//-------SIGNAL -> X_E_Tot_Cosu Max: 4.29497e+08 Min: 0 Def: 0 Resolution: 0.1 Offset: 0
GVL.IOVD.X_E_Tot_Cosu.v						:= GVL.SY.S_ECU_Rdy AND NOT GVL.IOVD.X_E_Tot_Cosu.e	AND NOT GVL.IOVD.X_E_Tot_Cosu.na AND NOT GVL.IOVD.X_E_Tot_Cosu.RangeExcd;
GVL.IOVD.X_E_Tot_Cosu.x						:= GVL.PV.X_E_Tot_Cosu;
GVL.IOVD.X_E_Tot_Cosu.e						:= FALSE;
GVL.IOVD.X_E_Tot_Cosu.na					:= FALSE;
GVL.IOVD.X_E_Tot_Cosu.RangeExcd				:= (429496729.4 < GVL.IOVD.X_E_Tot_Cosu.x) OR (0 > GVL.IOVD.X_E_Tot_Cosu.x);	 
//-------SIGNAL -> X_Avg_Cosu_Opp Max: 65,535 Min: 0 Def: 0 Resolution: 0.1 Offset: 0
GVL.IOVD.X_Avg_Cosu_Opp.v					:= GVL.SY.S_ECU_Rdy AND NOT GVL.IOVD.X_Avg_Cosu_Opp.e	AND NOT GVL.IOVD.X_Avg_Cosu_Opp.na AND NOT GVL.IOVD.X_Avg_Cosu_Opp.RangeExcd;
GVL.IOVD.X_Avg_Cosu_Opp.x					:= GVL.PV.X_Avg_Cosu_Opp;
GVL.IOVD.X_Avg_Cosu_Opp.e					:= FALSE;
GVL.IOVD.X_Avg_Cosu_Opp.na					:= FALSE;
GVL.IOVD.X_Avg_Cosu_Opp.RangeExcd			:= (65.535 < GVL.IOVD.X_Avg_Cosu_Opp.x) OR (0 > GVL.IOVD.X_Avg_Cosu_Opp.x);		  
{endregion}
//-----------------------------------------------------------------------------------------------------------------------------
//-----------------------------------------------------------------------------------------------------------------------------
//MESSAGE------
{region " User Area : Arac_Genel_Istatistik_2- ID:4C9"}

//-------SIGNAL -> X_Daily_Avg_Cosu Max: 40 Min: 0 Def: 0 Resolution: 0.001 Offset: 0
GVL.IOVD.X_Daily_Avg_Cosu.v					:= GVL.SY.S_ECU_Rdy AND NOT GVL.IOVD.X_Daily_Avg_Cosu.e	AND NOT GVL.IOVD.X_Daily_Avg_Cosu.na AND NOT GVL.IOVD.X_Daily_Avg_Cosu.RangeExcd;
GVL.IOVD.X_Daily_Avg_Cosu.x					:= GVL.PV.X_Avg_Cosu;
GVL.IOVD.X_Daily_Avg_Cosu.e					:= FALSE;
GVL.IOVD.X_Daily_Avg_Cosu.na				:= FALSE;
GVL.IOVD.X_Daily_Avg_Cosu.RangeExcd			:= (40 < GVL.IOVD.X_Daily_Avg_Cosu.x) OR (0 > GVL.IOVD.X_Daily_Avg_Cosu.x);
//-------SIGNAL -> X_Trp_Distn Max: 4.21108e+08 Min: 0 Def: 0 Resolution: 0.1 Offset: 0
GVL.IOVD.X_Trp_Distn.v						:= GVL.SY.S_ECU_Rdy AND NOT GVL.IOVD.X_Trp_Distn.e	AND NOT GVL.IOVD.X_Trp_Distn.na AND NOT GVL.IOVD.X_Trp_Distn.RangeExcd;
GVL.IOVD.X_Trp_Distn.x						:= GVL.PV.X_Trp_Bat;
GVL.IOVD.X_Trp_Distn.e						:= FALSE;
GVL.IOVD.X_Trp_Distn.na						:= FALSE;
GVL.IOVD.X_Trp_Distn.RangeExcd				:= (421108121.5 < GVL.IOVD.X_Trp_Distn.x) OR (0 > GVL.IOVD.X_Trp_Distn.x);
//-------SIGNAL -> X_U_ECU_Sp Max: 100 Min: 0 Def: 0 Resolution: 1 Offset: 0
GVL.IOVD.X_U_ECU_Sp.v						:= GVL.SY.S_ECU_Rdy AND NOT GVL.IOVD.X_U_ECU_Sp.e	AND NOT GVL.IOVD.X_U_ECU_Sp.na AND NOT GVL.IOVD.X_U_ECU_Sp.RangeExcd;
GVL.IOVD.X_U_ECU_Sp.x						:= ANY_TO_REAL(GVL.IC.X_U_Bat.value);
GVL.IOVD.X_U_ECU_Sp.e						:= FALSE;
GVL.IOVD.X_U_ECU_Sp.na						:= FALSE;
GVL.IOVD.X_U_ECU_Sp.RangeExcd				:= (40000 < GVL.IOVD.X_U_ECU_Sp.x )OR (0 > GVL.IOVD.X_U_ECU_Sp.x);		
{endregion}
//-----------------------------------------------------------------------------------------------------------------------------
//-----------------------------------------------------------------------------------------------------------------------------
//MESSAGE------
{region " User Area : Klima_Calisma_Sureleri_1- ID:4CA"}

//-------SIGNAL -> N_Hvac_Drv_Op_Cnt Max: 4.29497e+09 Min: 0 Def: 0 Resolution: 1 Offset: 0
GVL.IOVD.N_Hvac_Drv_Op_Cnt.v				:= GVL.SY.S_ECU_Rdy AND NOT GVL.IOVD.N_Hvac_Drv_Op_Cnt.e AND NOT GVL.IOVD.N_Hvac_Drv_Op_Cnt.na AND NOT GVL.IOVD.N_Hvac_Drv_Op_Cnt.RangeExcd;
GVL.IOVD.N_Hvac_Drv_Op_Cnt.x				:= DINT_TO_UDINT(TRUNC(GVL.PV.X_Tm_Tot_HVAC_Drv_Op / 60));		// PR1006_REV_002637_TIMTRO
GVL.IOVD.N_Hvac_Drv_Op_Cnt.e				:= FALSE;
GVL.IOVD.N_Hvac_Drv_Op_Cnt.na				:= FALSE;
GVL.IOVD.N_Hvac_Drv_Op_Cnt.RangeExcd		:= (4294967294 < GVL.IOVD.N_Hvac_Drv_Op_Cnt.x) OR (0 > GVL.IOVD.N_Hvac_Drv_Op_Cnt.x);
//-------SIGNAL -> N_Hvac_Pass1_Op_Cnt Max: 4.29497e+09 Min: 0 Def: 0 Resolution: 1 Offset: 0
GVL.IOVD.N_Hvac_Pass1_Op_Cnt.v				:= GVL.SY.S_ECU_Rdy AND NOT GVL.IOVD.N_Hvac_Pass1_Op_Cnt.e	AND NOT GVL.IOVD.N_Hvac_Pass1_Op_Cnt.na AND NOT GVL.IOVD.N_Hvac_Pass1_Op_Cnt.RangeExcd;
GVL.IOVD.N_Hvac_Pass1_Op_Cnt.x				:= DINT_TO_UDINT(TRUNC(GVL.PV.X_Tm_Tot_HVAC_Pass1_Op / 60));	// PR1006_REV_002637_TIMTRO
GVL.IOVD.N_Hvac_Pass1_Op_Cnt.e				:= FALSE;
GVL.IOVD.N_Hvac_Pass1_Op_Cnt.na				:= FALSE;
GVL.IOVD.N_Hvac_Pass1_Op_Cnt.RangeExcd		:= (4294967294 < GVL.IOVD.N_Hvac_Pass1_Op_Cnt.x) OR (0 > GVL.IOVD.N_Hvac_Pass1_Op_Cnt.x);
{endregion}
//-----------------------------------------------------------------------------------------------------------------------------
//-----------------------------------------------------------------------------------------------------------------------------
//MESSAGE------
{region " User Area : Klima_Calisma_Sureleri_2- ID:4CB"}

//-------SIGNAL -> N_Hvac_Pass2_Op_Cnt Max: 4.29497e+09 Min: 0 Def: 0 Resolution: 1 Offset: 0
GVL.IOVD.N_Hvac_Pass2_Op_Cnt.v				:= GVL.SY.S_ECU_Rdy AND NOT GVL.IOVD.N_Hvac_Pass2_Op_Cnt.e	AND NOT GVL.IOVD.N_Hvac_Pass2_Op_Cnt.na AND NOT GVL.IOVD.N_Hvac_Pass2_Op_Cnt.RangeExcd;
GVL.IOVD.N_Hvac_Pass2_Op_Cnt.x				:= T_N_Hvac_Pass2_Op_Cnt; //eklenecek
GVL.IOVD.N_Hvac_Pass2_Op_Cnt.e				:= FALSE;
GVL.IOVD.N_Hvac_Pass2_Op_Cnt.na				:= FALSE;
GVL.IOVD.N_Hvac_Pass2_Op_Cnt.RangeExcd		:= (4294967294 < GVL.IOVD.N_Hvac_Pass2_Op_Cnt.x) OR (0 > GVL.IOVD.N_Hvac_Pass2_Op_Cnt.x);
//-------SIGNAL -> N_Btms_Op_Cnt Max: 4.29497e+09 Min: 0 Def: 0 Resolution: 1 Offset: 0
GVL.IOVD.N_Btms_Op_Cnt.v					:= GVL.SY.S_ECU_Rdy AND NOT GVL.IOVD.N_Btms_Op_Cnt.e AND NOT GVL.IOVD.N_Btms_Op_Cnt.na AND NOT GVL.IOVD.N_Btms_Op_Cnt.RangeExcd;
GVL.IOVD.N_Btms_Op_Cnt.x					:= REAL_TO_UDINT(GVL.PV.X_Tm_Tot_BTMS_Op); // PR1006_REV_002446_TIMTRO
GVL.IOVD.N_Btms_Op_Cnt.e					:= FALSE;
GVL.IOVD.N_Btms_Op_Cnt.na					:= FALSE;
GVL.IOVD.N_Btms_Op_Cnt.RangeExcd			:= (4294967294 < GVL.IOVD.N_Btms_Op_Cnt.x) OR (0 > GVL.IOVD.N_Btms_Op_Cnt.x);
{endregion}
//-----------------------------------------------------------------------------------------------------------------------------
//-----------------------------------------------------------------------------------------------------------------------------
//MESSAGE------
{region " User Area : Sayicilar_1- ID:4CC"}

// PR1006_REV_002519_TIMTRO
//-------SIGNAL -> N_Air_Cmp_Op_Cnt Max: 4.29497e+09 Min: 0 Def: 0 Resolution: 1 Offset: 0
GVL.IOVD.N_Air_Cmp_Op_Cnt.v					:= GVL.SY.S_ECU_Rdy AND NOT GVL.IOVD.N_Air_Cmp_Op_Cnt.e	AND NOT GVL.IOVD.N_Air_Cmp_Op_Cnt.na AND NOT GVL.IOVD.N_Air_Cmp_Op_Cnt.RangeExcd;
GVL.IOVD.N_Air_Cmp_Op_Cnt.x					:= REAL_TO_UDINT(GVL.PV.X_Tm_Tot_Air_Cmp_Op);
GVL.IOVD.N_Air_Cmp_Op_Cnt.e					:= FALSE;
GVL.IOVD.N_Air_Cmp_Op_Cnt.na					:= FALSE;
GVL.IOVD.N_Air_Cmp_Op_Cnt.RangeExcd			:= (4294967294 < GVL.IOVD.N_Air_Cmp_Op_Cnt.x) OR (0 > GVL.IOVD.N_Air_Cmp_Op_Cnt.x);
//-------SIGNAL -> X_Opp_Dist_Bat Max: 6535.5 Min: 0 Def: 0 Resolution: 1 Offset: 0
GVL.IOVD.X_Opp_Dist_Bat.v					:= GVL.SY.S_ECU_Rdy AND NOT GVL.IOVD.X_Opp_Dist_Bat.e	AND NOT GVL.IOVD.X_Opp_Dist_Bat.na AND NOT GVL.IOVD.X_Opp_Dist_Bat.RangeExcd;
GVL.IOVD.X_Opp_Dist_Bat.x					:= GVL.PV.X_Opp_Dist_Bat;
GVL.IOVD.X_Opp_Dist_Bat.e					:= FALSE;
GVL.IOVD.X_Opp_Dist_Bat.na					:= FALSE;
GVL.IOVD.X_Opp_Dist_Bat.RangeExcd			:= (6553.5 < GVL.IOVD.X_Opp_Dist_Bat.x ) OR (0 > GVL.IOVD.X_Opp_Dist_Bat.x);	 		  
{endregion}
//-----------------------------------------------------------------------------------------------------------------------------
//-----------------------------------------------------------------------------------------------------------------------------
//MESSAGE------
{region " User Area : Yardimci_Tuketici_Enerjileri- ID:4CD"}

//-------SIGNAL -> X_E_Aux_Cons Max: 4.29497e+08 Min: 0 Def: 0 Resolution: 0.1 Offset: 0
GVL.IOVD.X_E_Aux_Cons.v						:= GVL.SY.S_ECU_Rdy AND NOT GVL.IOVD.X_E_Aux_Cons.e	AND NOT GVL.IOVD.X_E_Aux_Cons.na AND NOT GVL.IOVD.X_E_Aux_Cons.RangeExcd;
GVL.IOVD.X_E_Aux_Cons.x						:= (GVL.PV.X_E_Tot_Aux_AC + GVL.PV.X_E_Tot_Aux_DC + GVL.PV.X_E_Tot_Aux_DC_24V) / 100;
GVL.IOVD.X_E_Aux_Cons.e						:= FALSE;
GVL.IOVD.X_E_Aux_Cons.na					:= FALSE;
GVL.IOVD.X_E_Aux_Cons.RangeExcd				:= (429496729.4 < GVL.IOVD.X_E_Aux_Cons.x ) OR (0 > GVL.IOVD.X_E_Aux_Cons.x);
//-------SIGNAL -> X_E_Aux_Hvac_Cons Max: 4.29497e+08 Min: 0 Def: 0 Resolution: 0.1 Offset: 0
GVL.IOVD.X_E_Aux_Hvac_Cons.v				:= GVL.SY.S_ECU_Rdy AND NOT GVL.IOVD.X_E_Cosu.e	AND NOT GVL.IOVD.X_E_Cosu.na AND NOT GVL.IOVD.X_E_Cosu.RangeExcd;
GVL.IOVD.X_E_Aux_Hvac_Cons.x				:= GVL.PV.X_E_Tot_Aux_DC / 100;
GVL.IOVD.X_E_Aux_Hvac_Cons.e				:= FALSE;
GVL.IOVD.X_E_Aux_Hvac_Cons.na				:= FALSE;
GVL.IOVD.X_E_Aux_Hvac_Cons.RangeExcd		:= (429496729.4 < GVL.IOVD.X_E_Aux_Hvac_Cons.x ) OR (0 > GVL.IOVD.X_E_Aux_Hvac_Cons.x);
{endregion}
//-----------------------------------------------------------------------------------------------------------------------------
//-----------------------------------------------------------------------------------------------------------------------------
//-----------------------------------------------------------------------------------------------------------------------------
//MESSAGE------
{region " User Area : Kapi_Sayicilari_1- ID:4CE"}

//-------SIGNAL -> N_Dr1_Cycle Max: 4.29497e+09 Min: 0 Def: 0 Resolution: 1 Offset: 0
GVL.IOVD.N_Dr1_Cycle.v					:= GVL.SY.S_ECU_Rdy AND NOT GVL.IOVD.N_Dr1_Cycle.RangeExcd;
GVL.IOVD.N_Dr1_Cycle.x					:= GVL.PV.N_Dr1_Cyc;
GVL.IOVD.N_Dr1_Cycle.RangeExcd			:= (4294967294 < GVL.IOVD.N_Dr1_Cycle.x) OR (0 > GVL.IOVD.N_Dr1_Cycle.x);
//-------SIGNAL -> N_Dr2_Cycle Max: 4.29497e+09 Min: 0 Def: 0 Resolution: 1 Offset: 0
GVL.IOVD.N_Dr2_Cycle.v					:= GVL.SY.S_ECU_Rdy AND NOT GVL.IOVD.N_Dr2_Cycle.RangeExcd;
GVL.IOVD.N_Dr2_Cycle.x					:= GVL.PV.N_Dr2_Cyc;
GVL.IOVD.N_Dr2_Cycle.RangeExcd			:= (4294967294 < GVL.IOVD.N_Dr2_Cycle.x) OR (0 > GVL.IOVD.N_Dr2_Cycle.x);
{endregion}
//-----------------------------------------------------------------------------------------------------------------------------
//-----------------------------------------------------------------------------------------------------------------------------
//MESSAGE------
{region " User Area : Kapi_Sayicilari_2- ID:4CE"}

//-------SIGNAL -> N_Dr3_Cycle Max: 4.29497e+09 Min: 0 Def: 0 Resolution: 1 Offset: 0
GVL.IOVD.N_Dr3_Cycle.v					:= GVL.SY.S_ECU_Rdy AND NOT GVL.IOVD.N_Dr3_Cycle.RangeExcd;
GVL.IOVD.N_Dr3_Cycle.x					:= GVL.PV.N_Dr3_Cyc;
GVL.IOVD.N_Dr3_Cycle.RangeExcd			:= (4294967294 < GVL.IOVD.N_Dr3_Cycle.x) OR (0 > GVL.IOVD.N_Dr3_Cycle.x);
//-------SIGNAL -> N_Dr4_Cycle Max: 4.29497e+09 Min: 0 Def: 0 Resolution: 1 Offset: 0
GVL.IOVD.N_Dr4_Cycle.v					:= GVL.SY.S_ECU_Rdy AND NOT GVL.IOVD.N_Dr4_Cycle.RangeExcd;
GVL.IOVD.N_Dr4_Cycle.x					:= 0;
GVL.IOVD.N_Dr4_Cycle.RangeExcd			:= (4294967294 < GVL.IOVD.N_Dr4_Cycle.x) OR (0 > GVL.IOVD.N_Dr4_Cycle.x);
{endregion}
//-----------------------------------------------------------------------------------------------------------------------------
//-----------------------------------------------------------------------------------------------------------------------------
//MESSAGE------
{region " User Area : Sarj_Enerjisi- ID:4D0"}

//-------SIGNAL -> X_E_Chrg_Pan Max: 4.29497e+08 Min: 0 Def: 0 Resolution: 0.1 Offset: 0
GVL.IOVD.X_E_Chrg_Pan.v					:= GVL.SY.S_ECU_Rdy AND NOT GVL.IOVD.X_E_Chrg_Pan.RangeExcd;
GVL.IOVD.X_E_Chrg_Pan.x					:= GVL.PV.X_E_Pnt_Chrg_Cosu;
GVL.IOVD.X_E_Chrg_Pan.RangeExcd			:= (429496729.4 < GVL.IOVD.X_E_Chrg_Pan.x) OR (0 > GVL.IOVD.X_E_Chrg_Pan.x);
//-------SIGNAL -> X_E_Chrg_Onbrd Max: 4.29497e+08 Min: 0 Def: 0 Resolution: 0.1 Offset: 0
GVL.IOVD.X_E_Chrg_Onbrd.v				:= GVL.SY.S_ECU_Rdy AND NOT GVL.IOVD.X_E_Chrg_Onbrd.RangeExcd;
GVL.IOVD.X_E_Chrg_Onbrd.x				:= GVL.PV.X_E_Ser_Chrg_Cosu;
GVL.IOVD.X_E_Chrg_Onbrd.RangeExcd		:= (429496729.4 < GVL.IOVD.X_E_Chrg_Onbrd.x) OR (0 > GVL.IOVD.X_E_Chrg_Onbrd.x);
{endregion}
//-----------------------------------------------------------------------------------------------------------------------------
//-----------------------------------------------------------------------------------------------------------------------------

//MESSAGE------
{region " User Area : Arac_Bilgi_1- ID:4E0"}

//-------SIGNAL -> X_Vh_No Max: 65000 Min: 0 Def: 0 Resolution: 1 Offset: 0
GVL.IOVD.X_Vh_No.v						:= GVL.SY.S_ECU_Rdy AND NOT GVL.IOVD.X_Vh_No.e AND NOT GVL.IOVD.X_Vh_No.na AND NOT GVL.IOVD.X_Vh_No.RangeExcd;
GVL.IOVD.X_Vh_No.x						:= GVL.PV.X_Vh_No;
GVL.IOVD.X_Vh_No.e						:= FALSE;
GVL.IOVD.X_Vh_No.na						:= FALSE;
GVL.IOVD.X_Vh_No.RangeExcd				:= (65000 < GVL.IOVD.X_Vh_No.x) OR (0 > GVL.IOVD.X_Vh_No.x);
//-------SIGNAL -> X_Sw_Ver_Mjr_ECU Max: 250 Min: 0 Def: 0 Resolution: 1 Offset: 0
GVL.IOVD.X_Sw_Ver_Mjr_ECU.v				:= GVL.SY.S_ECU_Rdy AND NOT GVL.IOVD.X_Sw_Ver_Mjr_ECU.e	AND NOT GVL.IOVD.X_Sw_Ver_Mjr_ECU.na AND NOT GVL.IOVD.X_Sw_Ver_Mjr_ECU.RangeExcd;
GVL.IOVD.X_Sw_Ver_Mjr_ECU.x				:= GVL.IC.X_Sw_Ver_Mjr_ECU;
GVL.IOVD.X_Sw_Ver_Mjr_ECU.e				:= FALSE;
GVL.IOVD.X_Sw_Ver_Mjr_ECU.na			:= FALSE;
GVL.IOVD.X_Sw_Ver_Mjr_ECU.RangeExcd		:= (250 < GVL.IOVD.X_Sw_Ver_Mjr_ECU.x) OR (0 > GVL.IOVD.X_Sw_Ver_Mjr_ECU.x);
//-------SIGNAL -> X_Sw_Ver_Mnr_ECU Max: 250 Min: 0 Def: 0 Resolution: 1 Offset: 0
GVL.IOVD.X_Sw_Ver_Mnr_ECU.v				:= GVL.SY.S_ECU_Rdy AND NOT GVL.IOVD.X_Sw_Ver_Mnr_ECU.e	AND NOT GVL.IOVD.X_Sw_Ver_Mnr_ECU.na AND NOT GVL.IOVD.X_Sw_Ver_Mnr_ECU.RangeExcd;
GVL.IOVD.X_Sw_Ver_Mnr_ECU.x				:= GVL.IC.X_Sw_Ver_Mnr_ECU;
GVL.IOVD.X_Sw_Ver_Mnr_ECU.e				:= FALSE;
GVL.IOVD.X_Sw_Ver_Mnr_ECU.na			:= FALSE;
GVL.IOVD.X_Sw_Ver_Mnr_ECU.RangeExcd		:= (250 < GVL.IOVD.X_Sw_Ver_Mnr_ECU.x) OR (0 > GVL.IOVD.X_Sw_Ver_Mnr_ECU.x);
//-------SIGNAL -> X_Sw_Ver_Tst_ECU Max: 250 Min: 0 Def: 0 Resolution: 1 Offset: 0
GVL.IOVD.X_Sw_Ver_Tst_ECU.v				:= GVL.SY.S_ECU_Rdy AND NOT GVL.IOVD.X_Sw_Ver_Tst_ECU.e	AND NOT GVL.IOVD.X_Sw_Ver_Tst_ECU.na AND NOT GVL.IOVD.X_Sw_Ver_Tst_ECU.RangeExcd;
GVL.IOVD.X_Sw_Ver_Tst_ECU.x				:= GVL.IC.X_Sw_Ver_Tst_ECU;
GVL.IOVD.X_Sw_Ver_Tst_ECU.e				:= FALSE;
GVL.IOVD.X_Sw_Ver_Tst_ECU.na			:= FALSE;
GVL.IOVD.X_Sw_Ver_Tst_ECU.RangeExcd		:= (250 < GVL.IOVD.X_Sw_Ver_Tst_ECU.x) OR (0 > GVL.IOVD.X_Sw_Ver_Tst_ECU.x);
//-----------------------------------------------------------------------------------------------------------------------------
//-----------------------------------------------------------------------------------------------------------------------------
{region " MESSAGE AREA :HVAC_Sicaklik- ID:403"}

{region " SIGNAL AREA : NAME->S_ER_Susp_Amb LENGTH->1 STARTBIT :0"}
_FB_CanTx_Message_Unpack_403.S_Bit_0 	:= GVL.IOVD.S_ER_Susp_Amb;
{endregion}

{region " SIGNAL AREA : NAME->S_ER_Susp_Red LENGTH->1 STARTBIT :1"}
_FB_CanTx_Message_Unpack_403.S_Bit_1 	:= GVL.IOVD.S_ER_Susp_Red;
{endregion}

{region " SIGNAL AREA : NAME->S_ER_Lo_Pr_Amb LENGTH->1 STARTBIT :2"}
_FB_CanTx_Message_Unpack_403.S_Bit_2 	:= GVL.IOVD.S_ER_Lo_Pr_Amb;
{endregion}

{region " SIGNAL AREA : NAME->S_ER_Lo_Pr_Red LENGTH->1 STARTBIT :3"}
_FB_CanTx_Message_Unpack_403.S_Bit_3 	:= GVL.IOVD.S_ER_Lo_Pr_Red;
{endregion}

{region " SIGNAL AREA : NAME->S_ER_Ret LENGTH->1 STARTBIT :4"}
_FB_CanTx_Message_Unpack_403.S_Bit_4 	:= GVL.IOVD.S_ER_Ret;
{endregion}

{region " SIGNAL AREA : NAME->P_X_Tm_Dr_Cl_Rls LENGTH->8 STARTBIT :8"}
_FB_CanTx_Message_Unpack_403.X_Byte_1			:=
(*SELECT 1 : Is data valid and range is not exceed?*)	SEL((GVL.IOVD.P_X_Tm_Dr_Cl_Rls.v AND NOT GVL.IOVD.P_X_Tm_Dr_Cl_Rls.RangeExcd),
(*SELECT 2 : Is NOT AVAILABLE ?*)						SEL(GVL.IOVD.P_X_Tm_Dr_Cl_Rls.na,
(*SELECT 3 : Is ERROR active ?*)						SEL(GVL.IOVD.P_X_Tm_Dr_Cl_Rls.e,
(*DEFAULT VALUE assignment*)							0,
(*ERROR is active*)										16#FE),
(*NOT AVAILABLE is active*)								16#FF),
(*Transmission is VALID*)								USINT_TO_BYTE(REAL_TO_USINT((GVL.IOVD.P_X_Tm_Dr_Cl_Rls.x / 5))));			// PR1006_REV_002702_TIMTRO
{endregion}
			   
{region " SIGNAL AREA : NAME->P_X_Tm_Vld_ShtDn LENGTH->8 STARTBIT :16"}
_FB_CanTx_Message_Unpack_403.X_Byte_2			:=
(*SELECT 1 : Is data valid and range is not exceed?*)	SEL((GVL.IOVD.P_X_Tm_Vld_ShtDn.v AND NOT GVL.IOVD.P_X_Tm_Vld_ShtDn.RangeExcd),
(*SELECT 2 : Is NOT AVAILABLE ?*)						SEL(GVL.IOVD.P_X_Tm_Vld_ShtDn.na,
(*SELECT 3 : Is ERROR active ?*)						SEL(GVL.IOVD.P_X_Tm_Vld_ShtDn.e,
(*DEFAULT VALUE assignment*)							0,
(*ERROR is active*)										16#FE),
(*NOT AVAILABLE is active*)								16#FF),
(*Transmission is VALID*)								USINT_TO_BYTE(REAL_TO_USINT((GVL.IOVD.P_X_Tm_Vld_ShtDn.x / 5))));			// PR1006_REV_002702_TIMTRO
{endregion}	

{region " SIGNAL AREA : NAME->P_X_Tm_Lgt_Dr_ShtDn LENGTH->8 STARTBIT :24"}
_FB_CanTx_Message_Unpack_403.X_Byte_3			:=
(*SELECT 1 : Is data valid and range is not exceed?*)	SEL((GVL.IOVD.P_X_Tm_Lgt_Dr_ShtDn.v AND NOT GVL.IOVD.P_X_Tm_Lgt_Dr_ShtDn.RangeExcd),
(*SELECT 2 : Is NOT AVAILABLE ?*)						SEL(GVL.IOVD.P_X_Tm_Lgt_Dr_ShtDn.na,
(*SELECT 3 : Is ERROR active ?*)						SEL(GVL.IOVD.P_X_Tm_Lgt_Dr_ShtDn.e,
(*DEFAULT VALUE assignment*)							0,
(*ERROR is active*)										16#FE),
(*NOT AVAILABLE is active*)								16#FF),
(*Transmission is VALID*)								USINT_TO_BYTE(REAL_TO_USINT((GVL.IOVD.P_X_Tm_Lgt_Dr_ShtDn.x / 5))));		// PR1006_REV_002702_TIMTRO
{endregion}						 
	
_FB_CanTx_Message_Unpack_403.S_Bit_5 	:= TRUE;
_FB_CanTx_Message_Unpack_403.S_Bit_6 	:= TRUE;
_FB_CanTx_Message_Unpack_403.S_Bit_7 	:= TRUE;
_FB_CanTx_Message_Unpack_403.X_Byte_4 	:= 16#FF;
_FB_CanTx_Message_Unpack_403.X_Byte_5 	:= 16#FF;
_FB_CanTx_Message_Unpack_403.X_Byte_6 	:= 16#FF;
_FB_CanTx_Message_Unpack_403.X_Byte_7 	:= 16#FF;		
	
_FB_CanTx_Message_Unpack_403 (		C_Enable		:= GVL.IOVD.C_En_ECU_Parametre_0X403,
     								Obj_CAN			:= ADR(GVL.IC.Obj_CAN0),
     								X_MsgID			:= 16#403,
     								Tm_CycleTime	:= TIME#250MS,
     								N_Msg_Dlc		:= 8,
     								S_Extended		:= 0,
     								S_Sent_Ok   	=> GVL.IOVD.S_SentOk_ECU_Parametre_0X403);	  
{endregion}
//-----------------------------------------------------------------------------------------------------------------------------
//-----------------------------------------------------------------------------------------------------------------------------
{region " MESSAGE AREA :HVAC_Durum- ID:410"}

{region " SIGNAL AREA : NAME->S_HVAC_Sp LENGTH->2 STARTBIT :0"}
_FB_CanTx_Message_Unpack_410.S_Bit_0		:=	 (GVL.IOVD.S_HVAC_Sp.x OR GVL.IOVD.S_HVAC_Sp.na) AND NOT GVL.IOVD.S_HVAC_Sp.e; 
_FB_CanTx_Message_Unpack_410.S_Bit_1		:=	 NOT GVL.IOVD.S_HVAC_Sp.v OR GVL.IOVD.S_HVAC_Sp.na OR GVL.IOVD.S_HVAC_Sp.e; 
{endregion}

{region " SIGNAL AREA : NAME->S_HVAC_Mn_Swc LENGTH->2 STARTBIT :2"}
_FB_CanTx_Message_Unpack_410.S_Bit_2		:=	 (GVL.IOVD.S_HVAC_Mn_Swc.x OR GVL.IOVD.S_HVAC_Mn_Swc.na) AND NOT GVL.IOVD.S_HVAC_Mn_Swc.e; 
_FB_CanTx_Message_Unpack_410.S_Bit_3		:=	 NOT GVL.IOVD.S_HVAC_Mn_Swc.v OR GVL.IOVD.S_HVAC_Mn_Swc.na OR GVL.IOVD.S_HVAC_Mn_Swc.e; 
{endregion}

{region " SIGNAL AREA : NAME->S_HVAC_Otp_Do LENGTH->2 STARTBIT :4"}
_FB_CanTx_Message_Unpack_410.S_Bit_4		:=	 (GVL.IOVD.S_HVAC_Otp_Do.x OR GVL.IOVD.S_HVAC_Otp_Do.na) AND NOT GVL.IOVD.S_HVAC_Otp_Do.e; 
_FB_CanTx_Message_Unpack_410.S_Bit_5		:=	 NOT GVL.IOVD.S_HVAC_Otp_Do.v OR GVL.IOVD.S_HVAC_Otp_Do.na OR GVL.IOVD.S_HVAC_Otp_Do.e; 
{endregion}

{region " SIGNAL AREA : NAME->C_Dmst_On LENGTH->2 STARTBIT :6"}
_FB_CanTx_Message_Unpack_410.S_Bit_6		:=	 (GVL.IOVD.C_Dmst_On.x OR GVL.IOVD.C_Dmst_On.na) AND NOT GVL.IOVD.C_Dmst_On.e; 
_FB_CanTx_Message_Unpack_410.S_Bit_7		:=	 NOT GVL.IOVD.C_Dmst_On.v OR GVL.IOVD.C_Dmst_On.na OR GVL.IOVD.C_Dmst_On.e; 
{endregion}

{region " SIGNAL AREA : NAME->S_BTMS_En LENGTH->2 STARTBIT :8"}
_FB_CanTx_Message_Unpack_410.S_Bit_8		:=	 (GVL.IOVD.S_BTMS_En.x OR GVL.IOVD.S_BTMS_En.na) AND NOT GVL.IOVD.S_BTMS_En.e; 
_FB_CanTx_Message_Unpack_410.S_Bit_9		:=	 NOT GVL.IOVD.S_BTMS_En.v OR GVL.IOVD.S_BTMS_En.na OR GVL.IOVD.S_BTMS_En.e; 
{endregion}

{region " SIGNAL AREA : NAME->S_Elec_Heat_1_En LENGTH->2 STARTBIT :10"}
_FB_CanTx_Message_Unpack_410.S_Bit_10		:=	 (GVL.IOVD.S_Elec_Heat_1_En.x OR GVL.IOVD.S_Elec_Heat_1_En.na) AND NOT GVL.IOVD.S_Elec_Heat_1_En.e; 
_FB_CanTx_Message_Unpack_410.S_Bit_11		:=	 NOT GVL.IOVD.S_Elec_Heat_1_En.v OR GVL.IOVD.S_Elec_Heat_1_En.na OR GVL.IOVD.S_Elec_Heat_1_En.e; 
{endregion}

{region " SIGNAL AREA : NAME->S_Elec_Heat_2_En LENGTH->2 STARTBIT :12"}
_FB_CanTx_Message_Unpack_410.S_Bit_12		:=	 (GVL.IOVD.S_Elec_Heat_2_En.x OR GVL.IOVD.S_Elec_Heat_2_En.na) AND NOT GVL.IOVD.S_Elec_Heat_2_En.e; 
_FB_CanTx_Message_Unpack_410.S_Bit_13		:=	 NOT GVL.IOVD.S_Elec_Heat_2_En.v OR GVL.IOVD.S_Elec_Heat_2_En.na OR GVL.IOVD.S_Elec_Heat_2_En.e; 
{endregion}

{region " SIGNAL AREA : NAME->S_HVAC_Inver_En LENGTH->2 STARTBIT :14"}
_FB_CanTx_Message_Unpack_410.S_Bit_14		:=	 (GVL.IOVD.S_HVAC_Inver_En.x OR GVL.IOVD.S_HVAC_Inver_En.na) AND NOT GVL.IOVD.S_HVAC_Inver_En.e; 
_FB_CanTx_Message_Unpack_410.S_Bit_15		:=	 NOT GVL.IOVD.S_HVAC_Inver_En.v OR GVL.IOVD.S_HVAC_Inver_En.na OR GVL.IOVD.S_HVAC_Inver_En.e; 
{endregion}

{region " SIGNAL AREA : NAME->S_HVAC_1_En LENGTH->2 STARTBIT :16"}
_FB_CanTx_Message_Unpack_410.S_Bit_16		:=	 (GVL.IOVD.S_HVAC_1_En.x OR GVL.IOVD.S_HVAC_1_En.na) AND NOT GVL.IOVD.S_HVAC_1_En.e; 
_FB_CanTx_Message_Unpack_410.S_Bit_17		:=	 NOT GVL.IOVD.S_HVAC_1_En.v OR GVL.IOVD.S_HVAC_1_En.na OR GVL.IOVD.S_HVAC_1_En.e; 
{endregion}

{region " SIGNAL AREA : NAME->S_HVAC_2_En LENGTH->2 STARTBIT :18"}
_FB_CanTx_Message_Unpack_410.S_Bit_18		:=	 (GVL.IOVD.S_HVAC_2_En.x OR GVL.IOVD.S_HVAC_2_En.na) AND NOT GVL.IOVD.S_HVAC_2_En.e; 
_FB_CanTx_Message_Unpack_410.S_Bit_19		:=	 NOT GVL.IOVD.S_HVAC_2_En.v OR GVL.IOVD.S_HVAC_2_En.na OR GVL.IOVD.S_HVAC_2_En.e; 
{endregion}

{region " SIGNAL AREA : NAME->S_HVAC_Drv_En LENGTH->2 STARTBIT :20"}
_FB_CanTx_Message_Unpack_410.S_Bit_20		:=	 (GVL.IOVD.S_HVAC_Drv_En.x OR GVL.IOVD.S_HVAC_Drv_En.na) AND NOT GVL.IOVD.S_HVAC_Drv_En.e; 
_FB_CanTx_Message_Unpack_410.S_Bit_21		:=	 NOT GVL.IOVD.S_HVAC_Drv_En.v OR GVL.IOVD.S_HVAC_Drv_En.na OR GVL.IOVD.S_HVAC_Drv_En.e; 
{endregion}

{region " SIGNAL AREA : NAME->S_BTMS_Actv LENGTH->2 STARTBIT :24"}
_FB_CanTx_Message_Unpack_410.S_Bit_24		:=	 (GVL.IOVD.S_BTMS_Actv.x OR GVL.IOVD.S_BTMS_Actv.na) AND NOT GVL.IOVD.S_BTMS_Actv.e; 
_FB_CanTx_Message_Unpack_410.S_Bit_25		:=	 NOT GVL.IOVD.S_BTMS_Actv.v OR GVL.IOVD.S_BTMS_Actv.na OR GVL.IOVD.S_BTMS_Actv.e; 
{endregion}

{region " SIGNAL AREA : NAME->Z_BTMS_Mode LENGTH->2 STARTBIT :26"}
_FB_UNPACK_BYTE_TO_8BITS_4 ( 	S_Bit_0		=> _FB_CanTx_Message_Unpack_410.S_Bit_26,
								S_Bit_1		=> _FB_CanTx_Message_Unpack_410.S_Bit_27,
								X_BYTE_0	:=	GVL.IOVD.Z_BTMS_Mode.x);
{endregion}

{region " SIGNAL AREA : NAME->Z_BTMS_Req_Mode LENGTH->2 STARTBIT :28"}
_FB_UNPACK_BYTE_TO_8BITS_6 ( 	S_Bit_0		=> _FB_CanTx_Message_Unpack_410.S_Bit_28,
								S_Bit_1		=> _FB_CanTx_Message_Unpack_410.S_Bit_29,
								X_BYTE_0	:=
(*SELECT 1 : Is data valid and range is not exceed?*)	SEL((GVL.IOVD.Z_BTMS_Req_Mode.v AND NOT GVL.IOVD.Z_BTMS_Req_Mode.RangeExcd),
(*SELECT 2 : Is NOT AVAILABLE ?*)						SEL(GVL.IOVD.Z_BTMS_Req_Mode.na,
(*SELECT 3 : Is ERROR active ?*)						SEL(GVL.IOVD.Z_BTMS_Req_Mode.e,
(*DEFAULT VALUE assignment*)							0,
(*ERROR is active*)										16#E),
(*NOT AVAILABLE is active*)								16#F),
(*Transmission is VALID*)								GVL.IOVD.Z_BTMS_Req_Mode.x));
{endregion}

{region " SIGNAL AREA : NAME->S_Elec_Heat_1_On LENGTH->2 STARTBIT :30"}
_FB_CanTx_Message_Unpack_410.S_Bit_30		:=	 (GVL.IOVD.S_Elec_Heat_1_On.x OR GVL.IOVD.S_Elec_Heat_1_On.na) AND NOT GVL.IOVD.S_Elec_Heat_1_On.e; 
_FB_CanTx_Message_Unpack_410.S_Bit_31		:=	 NOT GVL.IOVD.S_Elec_Heat_1_On.v OR GVL.IOVD.S_Elec_Heat_1_On.na OR GVL.IOVD.S_Elec_Heat_1_On.e; 
{endregion}

{region " SIGNAL AREA : NAME->S_Elec_Heat_2_On LENGTH->2 STARTBIT :32"}
_FB_CanTx_Message_Unpack_410.S_Bit_32		:=	 (GVL.IOVD.S_Elec_Heat_2_On.x OR GVL.IOVD.S_Elec_Heat_2_On.na) AND NOT GVL.IOVD.S_Elec_Heat_2_On.e; 
_FB_CanTx_Message_Unpack_410.S_Bit_33		:=	 NOT GVL.IOVD.S_Elec_Heat_2_On.v OR GVL.IOVD.S_Elec_Heat_2_On.na OR GVL.IOVD.S_Elec_Heat_2_On.e; 
{endregion}

{region " SIGNAL AREA : NAME->S_HVAC_Inver_On LENGTH->2 STARTBIT :34"}
_FB_CanTx_Message_Unpack_410.S_Bit_34		:=	 (GVL.IOVD.S_HVAC_Inver_On.x OR GVL.IOVD.S_HVAC_Inver_On.na) AND NOT GVL.IOVD.S_HVAC_Inver_On.e; 
_FB_CanTx_Message_Unpack_410.S_Bit_35		:=	 NOT GVL.IOVD.S_HVAC_Inver_On.v OR GVL.IOVD.S_HVAC_Inver_On.na OR GVL.IOVD.S_HVAC_Inver_On.e; 
{endregion}

{region " SIGNAL AREA : NAME->S_Elec_Heat_Tm_On LENGTH->2 STARTBIT :36"}
_FB_CanTx_Message_Unpack_410.S_Bit_36		:=	 (GVL.IOVD.S_Elec_Heat_Tm_On.x OR GVL.IOVD.S_Elec_Heat_Tm_On.na) AND NOT GVL.IOVD.S_Elec_Heat_Tm_On.e; 
_FB_CanTx_Message_Unpack_410.S_Bit_37		:=	 NOT GVL.IOVD.S_Elec_Heat_Tm_On.v OR GVL.IOVD.S_Elec_Heat_Tm_On.na OR GVL.IOVD.S_Elec_Heat_Tm_On.e; 
{endregion}

{region " SIGNAL AREA : NAME->Z_HVAC_1_Mode LENGTH->4 STARTBIT :40"}
_FB_UNPACK_BYTE_TO_8BITS_0 ( 	S_Bit_0		=> _FB_CanTx_Message_Unpack_410.S_Bit_40,
								S_Bit_1		=> _FB_CanTx_Message_Unpack_410.S_Bit_41,
								S_Bit_2		=> _FB_CanTx_Message_Unpack_410.S_Bit_42,
								S_Bit_3		=> _FB_CanTx_Message_Unpack_410.S_Bit_43 ,
								X_BYTE_0	:=
(*SELECT 1 : Is data valid and range is not exceed?*)	SEL((GVL.IOVD.Z_HVAC_1_Mode.v AND NOT GVL.IOVD.Z_HVAC_1_Mode.RangeExcd),
(*SELECT 2 : Is NOT AVAILABLE ?*)						SEL(GVL.IOVD.Z_HVAC_1_Mode.na,
(*SELECT 3 : Is ERROR active ?*)						SEL(GVL.IOVD.Z_HVAC_1_Mode.e,
(*DEFAULT VALUE assignment*)							0,
(*ERROR is active*)										16#E),
(*NOT AVAILABLE is active*)								16#F),
(*Transmission is VALID*)								GVL.IOVD.Z_HVAC_1_Mode.x));
{endregion}

{region " SIGNAL AREA : NAME->Z_HVAC_2_Mode LENGTH->4 STARTBIT :44"}
_FB_UNPACK_BYTE_TO_8BITS_1 ( 	S_Bit_0		=> _FB_CanTx_Message_Unpack_410.S_Bit_44,
								S_Bit_1		=> _FB_CanTx_Message_Unpack_410.S_Bit_45,
								S_Bit_2		=> _FB_CanTx_Message_Unpack_410.S_Bit_46,
								S_Bit_3		=> _FB_CanTx_Message_Unpack_410.S_Bit_47 ,
								X_BYTE_0	:=
(*SELECT 1 : Is data valid and range is not exceed?*)	SEL((GVL.IOVD.Z_HVAC_2_Mode.v AND NOT GVL.IOVD.Z_HVAC_2_Mode.RangeExcd),
(*SELECT 2 : Is NOT AVAILABLE ?*)						SEL(GVL.IOVD.Z_HVAC_2_Mode.na,
(*SELECT 3 : Is ERROR active ?*)						SEL(GVL.IOVD.Z_HVAC_2_Mode.e,
(*DEFAULT VALUE assignment*)							0,
(*ERROR is active*)										16#E),
(*NOT AVAILABLE is active*)								16#F),
(*Transmission is VALID*)								GVL.IOVD.Z_HVAC_2_Mode.x));
{endregion}

{region " SIGNAL AREA : NAME->Z_HVAC_Drv_Mode LENGTH->4 STARTBIT :48"}
_FB_UNPACK_BYTE_TO_8BITS_2 ( 	S_Bit_0		=> _FB_CanTx_Message_Unpack_410.S_Bit_48,
								S_Bit_1		=> _FB_CanTx_Message_Unpack_410.S_Bit_49,
								S_Bit_2		=> _FB_CanTx_Message_Unpack_410.S_Bit_50,
								S_Bit_3		=> _FB_CanTx_Message_Unpack_410.S_Bit_51 ,
								X_BYTE_0	:=
(*SELECT 1 : Is data valid and range is not exceed?*)	SEL((GVL.IOVD.Z_HVAC_Drv_Mode.v AND NOT GVL.IOVD.Z_HVAC_Drv_Mode.RangeExcd),
(*SELECT 2 : Is NOT AVAILABLE ?*)						SEL(GVL.IOVD.Z_HVAC_Drv_Mode.na,
(*SELECT 3 : Is ERROR active ?*)						SEL(GVL.IOVD.Z_HVAC_Drv_Mode.e,
(*DEFAULT VALUE assignment*)							0,
(*ERROR is active*)										16#E),
(*NOT AVAILABLE is active*)								16#F),
(*Transmission is VALID*)								GVL.IOVD.Z_HVAC_Drv_Mode.x));
{endregion}

{region " SIGNAL AREA : NAME->Z_ER_HVAC LENGTH->4 STARTBIT :52"}
_FB_UNPACK_BYTE_TO_8BITS_3 ( 	S_Bit_0		=> _FB_CanTx_Message_Unpack_410.S_Bit_52,
								S_Bit_1		=> _FB_CanTx_Message_Unpack_410.S_Bit_53,
								S_Bit_2		=> _FB_CanTx_Message_Unpack_410.S_Bit_54,
								S_Bit_3		=> _FB_CanTx_Message_Unpack_410.S_Bit_55 ,
								X_BYTE_0	:=
(*SELECT 1 : Is data valid and range is not exceed?*)	SEL((GVL.IOVD.Z_ER_HVAC.v AND NOT GVL.IOVD.Z_ER_HVAC.RangeExcd),
(*SELECT 2 : Is NOT AVAILABLE ?*)						SEL(GVL.IOVD.Z_ER_HVAC.na,
(*SELECT 3 : Is ERROR active ?*)						SEL(GVL.IOVD.Z_ER_HVAC.e,
(*DEFAULT VALUE assignment*)							0,
(*ERROR is active*)										16#E),
(*NOT AVAILABLE is active*)								16#F),
(*Transmission is VALID*)								GVL.IOVD.Z_ER_HVAC.x));
{endregion}

{region " SIGNAL AREA : NAME->X_Spd_HVAC_Fan LENGTH->8 STARTBIT :56"}
_FB_CanTx_Message_Unpack_410.X_Byte_7		:=
(*SELECT 1 : Is data valid and range is not exceed?*)	SEL((GVL.IOVD.X_Spd_HVAC_Fan.v AND NOT GVL.IOVD.X_Spd_HVAC_Fan.RangeExcd),
(*SELECT 2 : Is NOT AVAILABLE ?*)						SEL(GVL.IOVD.X_Spd_HVAC_Fan.na,
(*SELECT 3 : Is ERROR active ?*)						SEL(GVL.IOVD.X_Spd_HVAC_Fan.e,
(*DEFAULT VALUE assignment*)							 0 ,
(*ERROR is active*)										16#FE),
(*NOT AVAILABLE is active*)								16#FF),
(*Transmission is VALID*)								USINT_TO_BYTE(REAL_TO_USINT((GVL.IOVD.X_Spd_HVAC_Fan.x))));
{endregion}

_FB_CanTx_Message_Unpack_410.S_Bit_22			:= TRUE;
_FB_CanTx_Message_Unpack_410.S_Bit_23			:= TRUE;
_FB_CanTx_Message_Unpack_410.S_Bit_38			:= TRUE;
_FB_CanTx_Message_Unpack_410.S_Bit_39			:= TRUE;

_FB_CanTx_Message_Unpack_410 ( 	C_Enable		:= GVL.IOVD.C_En_HVAC_Durum_0X410,
     							Obj_CAN			:= ADR(GVL.IC.Obj_CAN0),
     							X_MsgID			:= 16#410,
     							Tm_CycleTime	:= TIME#1000MS,
     							N_Msg_Dlc		:= 8,
     							S_Extended		:= 0,
     							S_Sent_Ok   	=> GVL.IOVD.S_SentOk_HVAC_Durum_0X410);
{endregion}
//-----------------------------------------------------------------------------------------------------------------------------
//-----------------------------------------------------------------------------------------------------------------------------
{region " MESSAGE AREA :HVAC_Sicaklik- ID:411"}

{region " SIGNAL AREA : NAME->X_T_Drv LENGTH->8 STARTBIT :0"}
_FB_CanTx_Message_411.X_Byte_0		:=
(*SELECT 1 : Is data valid and range is not exceed?*)	SEL((GVL.IOVD.X_T_Drv.v AND NOT GVL.IOVD.X_T_Drv.RangeExcd),
(*SELECT 2 : Is NOT AVAILABLE ?*)						SEL(GVL.IOVD.X_T_Drv.na,
(*SELECT 3 : Is ERROR active ?*)						SEL(GVL.IOVD.X_T_Drv.e,
(*DEFAULT VALUE assignment*)							USINT_TO_BYTE(REAL_TO_USINT((40))),
(*ERROR is active*)										16#FE),
(*NOT AVAILABLE is active*)								16#FF),
(*Transmission is VALID*)								USINT_TO_BYTE(REAL_TO_USINT((GVL.IOVD.X_T_Drv.x + 40))));
{endregion}
{region " SIGNAL AREA : NAME->W_T_Drv LENGTH->8 STARTBIT :8"}
_FB_CanTx_Message_411.X_Byte_1		:=
(*SELECT 1 : Is data valid and range is not exceed?*)	SEL((GVL.IOVD.W_T_Drv.v AND NOT GVL.IOVD.W_T_Drv.RangeExcd),
(*SELECT 2 : Is NOT AVAILABLE ?*)						SEL(GVL.IOVD.W_T_Drv.na,
(*SELECT 3 : Is ERROR active ?*)						SEL(GVL.IOVD.W_T_Drv.e,
(*DEFAULT VALUE assignment*)							USINT_TO_BYTE(REAL_TO_USINT((40))),
(*ERROR is active*)										16#FE),
(*NOT AVAILABLE is active*)								16#FF),
(*Transmission is VALID*)								USINT_TO_BYTE(REAL_TO_USINT((GVL.IOVD.W_T_Drv.x + 40))));
{endregion}
{region " SIGNAL AREA : NAME->X_T_Insd_1 LENGTH->8 STARTBIT :16"}
_FB_CanTx_Message_411.X_Byte_2		:=
(*SELECT 1 : Is data valid and range is not exceed?*)	SEL((GVL.IOVD.X_T_Insd_1.v AND NOT GVL.IOVD.X_T_Insd_1.RangeExcd),
(*SELECT 2 : Is NOT AVAILABLE ?*)						SEL(GVL.IOVD.X_T_Insd_1.na,
(*SELECT 3 : Is ERROR active ?*)						SEL(GVL.IOVD.X_T_Insd_1.e,
(*DEFAULT VALUE assignment*)							USINT_TO_BYTE(REAL_TO_USINT((0))),
(*ERROR is active*)										16#FE),
(*NOT AVAILABLE is active*)								16#FF),
(*Transmission is VALID*)								USINT_TO_BYTE(REAL_TO_USINT((GVL.IOVD.X_T_Insd_1.x + 40))));
{endregion}
{region " SIGNAL AREA : NAME->X_T_Insd_2 LENGTH->8 STARTBIT :24"}
_FB_CanTx_Message_411.X_Byte_3		:=
(*SELECT 1 : Is data valid and range is not exceed?*)	SEL((GVL.IOVD.X_T_Insd_2.v AND NOT GVL.IOVD.X_T_Insd_2.RangeExcd),
(*SELECT 2 : Is NOT AVAILABLE ?*)						SEL(GVL.IOVD.X_T_Insd_2.na,
(*SELECT 3 : Is ERROR active ?*)						SEL(GVL.IOVD.X_T_Insd_2.e,
(*DEFAULT VALUE assignment*)							USINT_TO_BYTE(REAL_TO_USINT((0))),
(*ERROR is active*)										16#FE),
(*NOT AVAILABLE is active*)								16#FF),
(*Transmission is VALID*)								USINT_TO_BYTE(REAL_TO_USINT((GVL.IOVD.X_T_Insd_2.x + 40))));
{endregion}
{region " SIGNAL AREA : NAME->W_T_HVAC_Psng LENGTH->8 STARTBIT :32"}
_FB_CanTx_Message_411.X_Byte_4		:=
(*SELECT 1 : Is data valid and range is not exceed?*)	SEL((GVL.IOVD.W_T_HVAC_Psng.v AND NOT GVL.IOVD.W_T_HVAC_Psng.RangeExcd),
(*SELECT 2 : Is NOT AVAILABLE ?*)						SEL(GVL.IOVD.W_T_HVAC_Psng.na,
(*SELECT 3 : Is ERROR active ?*)						SEL(GVL.IOVD.W_T_HVAC_Psng.e,
(*DEFAULT VALUE assignment*)							USINT_TO_BYTE(REAL_TO_USINT((40))),
(*ERROR is active*)										16#FE),
(*NOT AVAILABLE is active*)								16#FF),
(*Transmission is VALID*)								USINT_TO_BYTE(REAL_TO_USINT((GVL.IOVD.W_T_HVAC_Psng.x + 40))));
{endregion}
{region " SIGNAL AREA : NAME->X_T_Amb LENGTH->8 STARTBIT :40"}
_FB_CanTx_Message_411.X_Byte_5		:=
(*SELECT 1 : Is data valid and range is not exceed?*)	SEL((GVL.IOVD.X_T_Amb.v AND NOT GVL.IOVD.X_T_Amb.RangeExcd),
(*SELECT 2 : Is NOT AVAILABLE ?*)						SEL(GVL.IOVD.X_T_Amb.na,
(*SELECT 3 : Is ERROR active ?*)						SEL(GVL.IOVD.X_T_Amb.e,
(*DEFAULT VALUE assignment*)							USINT_TO_BYTE(REAL_TO_USINT((40))),
(*ERROR is active*)										16#FE),
(*NOT AVAILABLE is active*)								16#FF),
(*Transmission is VALID*)								USINT_TO_BYTE(REAL_TO_USINT((GVL.IOVD.X_T_Amb.x + 40))));
{endregion}
{region " SIGNAL AREA : NAME->X_T_Clt_Wtr LENGTH->8 STARTBIT :48"}
_FB_CanTx_Message_411.X_Byte_6		:=
(*SELECT 1 : Is data valid and range is not exceed?*)	SEL((GVL.IOVD.X_T_Clt_Wtr.v AND NOT GVL.IOVD.X_T_Clt_Wtr.RangeExcd),
(*SELECT 2 : Is NOT AVAILABLE ?*)						SEL(GVL.IOVD.X_T_Clt_Wtr.na,
(*SELECT 3 : Is ERROR active ?*)						SEL(GVL.IOVD.X_T_Clt_Wtr.e,
(*DEFAULT VALUE assignment*)							USINT_TO_BYTE(REAL_TO_USINT((40))),
(*ERROR is active*)										16#FE),
(*NOT AVAILABLE is active*)								16#FF),
(*Transmission is VALID*)								USINT_TO_BYTE(REAL_TO_USINT((GVL.IOVD.X_T_Clt_Wtr.x + 40))));
{endregion}

_FB_CanTx_Message_411.X_Byte_7				:= 16#FF;

_FB_CanTx_Message_411 ( 	C_Enable		:= GVL.IOVD.C_En_HVAC_Sicaklik_0X411,
     						Obj_CAN			:= ADR(GVL.IC.Obj_CAN0),
     						X_MsgID			:= 16#411,
     						Tm_CycleTime	:= TIME#1000MS,
     						N_Msg_Dlc		:=8,
     						S_Extended		:= 0,
     						S_Sent_Ok  		=> GVL.IOVD.S_SentOk_HVAC_Sicaklik_0X411);
{endregion}
//-----------------------------------------------------------------------------------------------------------------------------
//-----------------------------------------------------------------------------------------------------------------------------
{region " MESSAGE AREA :HVAC_Analog- ID:413"}

{region " SIGNAL AREA : NAME->X_P_HVAC_Inver LENGTH->16 STARTBIT :0"}
_FB_UNPACK_WORD_TO_BYTE_0 ( 	X_WORD_0	:= 
(*SELECT 1 : Is data valid and range is not exceed?*)	SEL((GVL.IOVD.X_P_HVAC_Inver.v AND NOT GVL.IOVD.X_P_HVAC_Inver.RangeExcd),
(*SELECT 2 : Is NOT AVAILABLE ?*)						SEL(GVL.IOVD.X_P_HVAC_Inver.na,
(*SELECT 3 : Is ERROR active ?*)						SEL(GVL.IOVD.X_P_HVAC_Inver.e,
(*DEFAULT VALUE assignment*)							0,
(*ERROR is active*)										16#FEFE),
(*NOT AVAILABLE is active*)								16#FFFF),
(*Transmission is VALID*)								UINT_TO_WORD(REAL_TO_UINT((GVL.IOVD.X_P_HVAC_Inver.x)))),
								X_BYTE_0	=> _FB_CanTx_Message_413.X_Byte_0,
								X_BYTE_1	=> _FB_CanTx_Message_413.X_Byte_1);
{endregion}

{region " SIGNAL AREA : NAME->X_P_Elec_Heat LENGTH->16 STARTBIT :16"}
_FB_UNPACK_WORD_TO_BYTE_1 ( 	X_WORD_0	:= 
(*SELECT 1 : Is data valid and range is not exceed?*)	SEL((GVL.IOVD.X_P_Elec_Heat.v AND NOT GVL.IOVD.X_P_Elec_Heat.RangeExcd),
(*SELECT 2 : Is NOT AVAILABLE ?*)						SEL(GVL.IOVD.X_P_Elec_Heat.na,
(*SELECT 3 : Is ERROR active ?*)						SEL(GVL.IOVD.X_P_Elec_Heat.e,
(*DEFAULT VALUE assignment*)							0,
(*ERROR is active*)										16#FEFE),
(*NOT AVAILABLE is active*)								16#FFFF),
(*Transmission is VALID*)								UINT_TO_WORD(REAL_TO_UINT((GVL.IOVD.X_P_Elec_Heat.x)))),
								X_BYTE_0	=> _FB_CanTx_Message_413.X_Byte_2,
								X_BYTE_1	=> _FB_CanTx_Message_413.X_Byte_3);
{endregion}

{region " SIGNAL AREA : NAME->X_I_In_HVAC_Inver LENGTH->16 STARTBIT :32"}
_FB_UNPACK_WORD_TO_BYTE_2 (		X_WORD_0	:= 
(*SELECT 1 : Is data valid and range is not exceed?*)	SEL((GVL.IOVD.X_I_In_HVAC_Inver.v AND NOT GVL.IOVD.X_I_In_HVAC_Inver.RangeExcd),
(*SELECT 2 : Is NOT AVAILABLE ?*)						SEL(GVL.IOVD.X_I_In_HVAC_Inver.na,
(*SELECT 3 : Is ERROR active ?*)						SEL(GVL.IOVD.X_I_In_HVAC_Inver.e,
(*DEFAULT VALUE assignment*)							0,
(*ERROR is active*)										16#FEFE),
(*NOT AVAILABLE is active*)								16#FFFF),
(*Transmission is VALID*)								UINT_TO_WORD(REAL_TO_UINT((GVL.IOVD.X_I_In_HVAC_Inver.x) / 0.05))),
								X_BYTE_0	=> _FB_CanTx_Message_413.X_Byte_4,
								X_BYTE_1	=> _FB_CanTx_Message_413.X_Byte_5);
{endregion}

{region " SIGNAL AREA : NAME->X_I_In_Elec_Heat LENGTH->16 STARTBIT :48"}
_FB_UNPACK_WORD_TO_BYTE_3 ( 	X_WORD_0	:= 
(*SELECT 1 : Is data valid and range is not exceed?*)	SEL((GVL.IOVD.X_I_In_Elec_Heat.v AND NOT GVL.IOVD.X_I_In_Elec_Heat.RangeExcd),
(*SELECT 2 : Is NOT AVAILABLE ?*)						SEL(GVL.IOVD.X_I_In_Elec_Heat.na,
(*SELECT 3 : Is ERROR active ?*)						SEL(GVL.IOVD.X_I_In_Elec_Heat.e,
(*DEFAULT VALUE assignment*)							0,
(*ERROR is active*)										16#FEFE),
(*NOT AVAILABLE is active*)								16#FFFF),
(*Transmission is VALID*)								UINT_TO_WORD(REAL_TO_UINT((GVL.IOVD.X_I_In_Elec_Heat.x) / 0.05))),
								X_BYTE_0	=> _FB_CanTx_Message_413.X_Byte_6,
								X_BYTE_1	=> _FB_CanTx_Message_413.X_Byte_7);
{endregion}

_FB_CanTx_Message_413 ( 	C_Enable		:= GVL.IOVD.C_En_HVAC_Analog_0X413,
     						Obj_CAN			:= ADR(GVL.IC.Obj_CAN0),
     						X_MsgID			:= 16#413,
     						Tm_CycleTime	:= TIME#1000MS,
     						N_Msg_Dlc		:= 8,
     						S_Extended		:= 0,
     						S_Sent_Ok   	=> GVL.IOVD.S_SentOk_HVAC_Analog_0X413);
{endregion}
//-----------------------------------------------------------------------------------------------------------------------------
//-----------------------------------------------------------------------------------------------------------------------------
{region " MESSAGE AREA :Klima_Kontaktor_Kontrol- ID:414"}
{region " SIGNAL AREA : NAME->C_Defrs_Plus_Ct LENGTH->1 STARTBIT :0"}
_FB_CanTx_Message_Unpack_414.S_Bit_0				:= GVL.IOVD.C_Defrs_Plus_Ct.x AND GVL.IOVD.C_Defrs_Plus_Ct.v;
{endregion}
{region " SIGNAL AREA : NAME->C_Defrs_Minus_Ct LENGTH->1 STARTBIT :1"}
_FB_CanTx_Message_Unpack_414.S_Bit_1				:= GVL.IOVD.C_Defrs_Minus_Ct.x AND GVL.IOVD.C_Defrs_Minus_Ct.v;
{endregion}
{region " SIGNAL AREA : NAME->C_Prheat_Plus_Ct LENGTH->1 STARTBIT :2"}
_FB_CanTx_Message_Unpack_414.S_Bit_2				:= GVL.IOVD.C_Prheat_Plus_Ct.x AND GVL.IOVD.C_Prheat_Plus_Ct.v;
{endregion}
{region " SIGNAL AREA : NAME->C_Prheat_Minus_Ct LENGTH->1 STARTBIT :3"}
_FB_CanTx_Message_Unpack_414.S_Bit_3				:= GVL.IOVD.C_Prheat_Minus_Ct.x AND GVL.IOVD.C_Prheat_Minus_Ct.v;
{endregion}
{region " SIGNAL AREA : NAME->C_HVAC_Plus_Ct LENGTH->1 STARTBIT :4"}
_FB_CanTx_Message_Unpack_414.S_Bit_4				:= GVL.IOVD.C_HVAC_Plus_Ct.x AND GVL.IOVD.C_HVAC_Plus_Ct.v;
{endregion}
{region " SIGNAL AREA : NAME->C_HVAC_Minus_Ct LENGTH->1 STARTBIT :5"}
_FB_CanTx_Message_Unpack_414.S_Bit_5				:= GVL.IOVD.C_HVAC_Minus_Ct.x AND GVL.IOVD.C_HVAC_Minus_Ct.v;
{endregion}
{region " SIGNAL AREA : NAME->S_Defrs_Plus_Ct_Deactv LENGTH->1 STARTBIT :6"}
_FB_CanTx_Message_Unpack_414.S_Bit_6				:= GVL.IOVD.S_Defrs_Plus_Ct_Deactv.x AND GVL.IOVD.S_Defrs_Plus_Ct_Deactv.v;
{endregion}
{region " SIGNAL AREA : NAME->S_Defrs_Minus_Ct_Deactv LENGTH->1 STARTBIT :7"}
_FB_CanTx_Message_Unpack_414.S_Bit_7				:= GVL.IOVD.S_Defrs_Minus_Ct_Deactv.x AND GVL.IOVD.S_Defrs_Minus_Ct_Deactv.v;
{endregion}
{region " SIGNAL AREA : NAME->S_Prheat_Plus_Ct_Deactv LENGTH->1 STARTBIT :8"}
_FB_CanTx_Message_Unpack_414.S_Bit_8				:= GVL.IOVD.S_Prheat_Plus_Ct_Deactv.x AND GVL.IOVD.S_Prheat_Plus_Ct_Deactv.v;
{endregion}
{region " SIGNAL AREA : NAME->S_Prheat_Minus_Ct_Deactv LENGTH->1 STARTBIT :9"}
_FB_CanTx_Message_Unpack_414.S_Bit_9				:= GVL.IOVD.S_Prheat_Minus_Ct_Deactv.x AND GVL.IOVD.S_Prheat_Minus_Ct_Deactv.v;
{endregion}
{region " SIGNAL AREA : NAME->S_HVAC_Plus_Ct_Deactv LENGTH->1 STARTBIT :10"}
_FB_CanTx_Message_Unpack_414.S_Bit_10				:= GVL.IOVD.S_HVAC_Plus_Ct_Deactv.x AND GVL.IOVD.S_HVAC_Plus_Ct_Deactv.v;
{endregion}
{region " SIGNAL AREA : NAME->S_HVAC_Minus_Ct_Deactv LENGTH->1 STARTBIT :11"}
_FB_CanTx_Message_Unpack_414.S_Bit_11				:= GVL.IOVD.S_HVAC_Minus_Ct_Deactv.x AND GVL.IOVD.S_HVAC_Minus_Ct_Deactv.v;
{endregion}
{region " SIGNAL AREA : NAME->Z_Btms_Stat LENGTH->4 STARTBIT :12"}
_FB_UNPACK_BYTE_TO_8BITS_5 ( 	S_Bit_0		=> _FB_CanTx_Message_Unpack_414.S_Bit_12,
								S_Bit_1		=> _FB_CanTx_Message_Unpack_414.S_Bit_13,
								S_Bit_2		=> _FB_CanTx_Message_Unpack_414.S_Bit_14,
								S_Bit_3		=> _FB_CanTx_Message_Unpack_414.S_Bit_15 ,
								X_BYTE_0	:=
(*SELECT 1 : Is data valid and range is not exceed?*)	SEL((GVL.IOVD.Z_Btms_Stat.v AND NOT GVL.IOVD.Z_Btms_Stat.RangeExcd),
(*SELECT 2 : Is NOT AVAILABLE ?*)						SEL(GVL.IOVD.Z_Btms_Stat.na,
(*SELECT 3 : Is ERROR active ?*)						SEL(GVL.IOVD.Z_Btms_Stat.e,
(*DEFAULT VALUE assignment*)							0,
(*ERROR is active*)										16#E),
(*NOT AVAILABLE is active*)								16#F),
(*Transmission is VALID*)								GVL.IOVD.Z_Btms_Stat.x));
{endregion}
{region " SIGNAL AREA : NAME->Z_HvacDrv_Stat LENGTH->8 STARTBIT :16"}
_FB_CanTx_Message_Unpack_414.X_Byte_2		:=
(*SELECT 1 : Is data valid and range is not exceed?*)	SEL((GVL.IOVD.Z_HvacDrv_Stat.v AND NOT GVL.IOVD.Z_HvacDrv_Stat.RangeExcd),
(*SELECT 2 : Is NOT AVAILABLE ?*)						SEL(GVL.IOVD.Z_HvacDrv_Stat.na,
(*SELECT 3 : Is ERROR active ?*)						SEL(GVL.IOVD.Z_HvacDrv_Stat.e,
(*DEFAULT VALUE assignment*)							0,
(*ERROR is active*)										16#FE),
(*NOT AVAILABLE is active*)								16#FF),
(*Transmission is VALID*)								USINT_TO_BYTE(REAL_TO_USINT((GVL.IOVD.Z_HvacDrv_Stat.x))));
{endregion}
{region " SIGNAL AREA : NAME->Z_HvacDrv_Stat LENGTH->8 STARTBIT :24"}
_FB_CanTx_Message_Unpack_414.X_Byte_3		:=
(*SELECT 1 : Is data valid and range is not exceed?*)	SEL((GVL.IOVD.Z_HvacPass1_Stat.v AND NOT GVL.IOVD.Z_HvacPass1_Stat.RangeExcd),
(*SELECT 2 : Is NOT AVAILABLE ?*)						SEL(GVL.IOVD.Z_HvacPass1_Stat.na,
(*SELECT 3 : Is ERROR active ?*)						SEL(GVL.IOVD.Z_HvacPass1_Stat.e,
(*DEFAULT VALUE assignment*)							0,
(*ERROR is active*)										16#FE),
(*NOT AVAILABLE is active*)								16#FF),
(*Transmission is VALID*)								USINT_TO_BYTE(REAL_TO_USINT((GVL.IOVD.Z_HvacPass1_Stat.x))));
{endregion}
{region " SIGNAL AREA : NAME->Z_HvacDrv_Stat LENGTH->8 STARTBIT :32"}
_FB_CanTx_Message_Unpack_414.X_Byte_4		:=
(*SELECT 1 : Is data valid and range is not exceed?*)	SEL((GVL.IOVD.Z_HvacPass2_Stat.v AND NOT GVL.IOVD.Z_HvacPass2_Stat.RangeExcd),
(*SELECT 2 : Is NOT AVAILABLE ?*)						SEL(GVL.IOVD.Z_HvacPass2_Stat.na,
(*SELECT 3 : Is ERROR active ?*)						SEL(GVL.IOVD.Z_HvacPass2_Stat.e,
(*DEFAULT VALUE assignment*)							0,
(*ERROR is active*)										16#FE),
(*NOT AVAILABLE is active*)								16#FF),
(*Transmission is VALID*)								USINT_TO_BYTE(REAL_TO_USINT((GVL.IOVD.Z_HvacPass2_Stat.x))));
{endregion}
{region " SIGNAL AREA : NAME->Z_HvacDrv_Stat LENGTH->8 STARTBIT :40"}  
_FB_CanTx_Message_Unpack_414.X_Byte_5		:=
(*SELECT 1 : Is data valid and range is not exceed?*)	SEL((GVL.IOVD.Z_Elec_Heaters_Stat.v AND NOT GVL.IOVD.Z_Elec_Heaters_Stat.RangeExcd),
(*SELECT 2 : Is NOT AVAILABLE ?*)						SEL(GVL.IOVD.Z_Elec_Heaters_Stat.na,
(*SELECT 3 : Is ERROR active ?*)						SEL(GVL.IOVD.Z_Elec_Heaters_Stat.e,
(*DEFAULT VALUE assignment*)							0,
(*ERROR is active*)										16#FE),
(*NOT AVAILABLE is active*)								16#FF),
(*Transmission is VALID*)								USINT_TO_BYTE(REAL_TO_USINT((GVL.IOVD.Z_Elec_Heaters_Stat.x))));
{endregion}
{region " SIGNAL AREA : NAME->Z_HvacDrv_Stat LENGTH->8 STARTBIT :48"}  
_FB_CanTx_Message_Unpack_414.X_Byte_6		:=
(*SELECT 1 : Is data valid and range is not exceed?*)	SEL((GVL.IOVD.Z_Flr_Heaters_Stat_1.v AND NOT GVL.IOVD.Z_Flr_Heaters_Stat_1.RangeExcd),
(*SELECT 2 : Is NOT AVAILABLE ?*)						SEL(GVL.IOVD.Z_Flr_Heaters_Stat_1.na,
(*SELECT 3 : Is ERROR active ?*)						SEL(GVL.IOVD.Z_Flr_Heaters_Stat_1.e,
(*DEFAULT VALUE assignment*)							0,
(*ERROR is active*)										16#FE),
(*NOT AVAILABLE is active*)								16#FF),
(*Transmission is VALID*)								USINT_TO_BYTE(REAL_TO_USINT((GVL.IOVD.Z_Flr_Heaters_Stat_1.x))));
{endregion}
{region " SIGNAL AREA : NAME->Z_HvacDrv_Stat LENGTH->8 STARTBIT :56"}  
_FB_CanTx_Message_Unpack_414.X_Byte_7		:=
(*SELECT 1 : Is data valid and range is not exceed?*)	SEL((GVL.IOVD.Z_Flr_Heaters_Stat_2.v AND NOT GVL.IOVD.Z_Flr_Heaters_Stat_2.RangeExcd),
(*SELECT 2 : Is NOT AVAILABLE ?*)						SEL(GVL.IOVD.Z_Flr_Heaters_Stat_2.na,
(*SELECT 3 : Is ERROR active ?*)						SEL(GVL.IOVD.Z_Flr_Heaters_Stat_2.e,
(*DEFAULT VALUE assignment*)							0,
(*ERROR is active*)										16#FE),
(*NOT AVAILABLE is active*)								16#FF),
(*Transmission is VALID*)								USINT_TO_BYTE(REAL_TO_USINT((GVL.IOVD.Z_Flr_Heaters_Stat_2.x))));
{endregion}

_FB_CanTx_Message_Unpack_414 ( 	C_Enable		:= GVL.IOVD.C_En_Klima_Kontaktor_Kontrol_0X414,
     							Obj_CAN			:= ADR(GVL.IC.Obj_CAN0),
     							X_MsgID			:= 16#414,
     							Tm_CycleTime	:= TIME#1000MS,
     							N_Msg_Dlc		:= 8,
     							S_Extended		:= 0,
     							S_Sent_Ok   	=> GVL.IOVD.S_SentOk_Klima_Kontaktor_Kontrol_0X414);
{endregion}
//-----------------------------------------------------------------------------------------------------------------------------
//-----------------------------------------------------------------------------------------------------------------------------
{region " MESSAGE AREA :HVAC_Parameters_1- ID:415"}

{region " SIGNAL AREA : NAME->P_X_T_Max_Bat_BTMS_Heat LENGTH->8 STARTBIT :0"}
_FB_CanTx_Message_Unpack_415.X_Byte_0			:=
(*SELECT 1 : Is data valid and range is not exceed?*)	SEL((GVL.IOVD.P_X_T_Max_Bat_BTMS_Heat.v AND NOT GVL.IOVD.P_X_T_Max_Bat_BTMS_Heat.RangeExcd),
(*SELECT 2 : Is NOT AVAILABLE ?*)						SEL(GVL.IOVD.P_X_T_Max_Bat_BTMS_Heat.na,
(*SELECT 3 : Is ERROR active ?*)						SEL(GVL.IOVD.P_X_T_Max_Bat_BTMS_Heat.e,
(*DEFAULT VALUE assignment*)							0,
(*ERROR is active*)										16#FE),
(*NOT AVAILABLE is active*)								16#FF),
(*Transmission is VALID*)								USINT_TO_BYTE(REAL_TO_USINT((GVL.IOVD.P_X_T_Max_Bat_BTMS_Heat.x))));
{endregion}

{region " SIGNAL AREA : NAME->P_X_T_Max_Bat_BTMS_Cool LENGTH->8 STARTBIT :8"}
_FB_CanTx_Message_Unpack_415.X_Byte_1			:=
(*SELECT 1 : Is data valid and range is not exceed?*)	SEL((GVL.IOVD.P_X_T_Max_Bat_BTMS_Cool.v AND NOT GVL.IOVD.P_X_T_Max_Bat_BTMS_Cool.RangeExcd),
(*SELECT 2 : Is NOT AVAILABLE ?*)						SEL(GVL.IOVD.P_X_T_Max_Bat_BTMS_Cool.na,
(*SELECT 3 : Is ERROR active ?*)						SEL(GVL.IOVD.P_X_T_Max_Bat_BTMS_Cool.e,
(*DEFAULT VALUE assignment*)							0,
(*ERROR is active*)										16#FE),
(*NOT AVAILABLE is active*)								16#FF),
(*Transmission is VALID*)								USINT_TO_BYTE(REAL_TO_USINT((GVL.IOVD.P_X_T_Max_Bat_BTMS_Cool.x))));
{endregion}

{region " SIGNAL AREA : NAME->P_X_T_Max_Wtr_BTMS_Heat LENGTH->8 STARTBIT :16"}
_FB_CanTx_Message_Unpack_415.X_Byte_2			:=
(*SELECT 1 : Is data valid and range is not exceed?*)	SEL((GVL.IOVD.P_X_T_Max_Wtr_BTMS_Heat.v AND NOT GVL.IOVD.P_X_T_Max_Wtr_BTMS_Heat.RangeExcd),
(*SELECT 2 : Is NOT AVAILABLE ?*)						SEL(GVL.IOVD.P_X_T_Max_Wtr_BTMS_Heat.na,
(*SELECT 3 : Is ERROR active ?*)						SEL(GVL.IOVD.P_X_T_Max_Wtr_BTMS_Heat.e,
(*DEFAULT VALUE assignment*)							0,
(*ERROR is active*)										16#FE),
(*NOT AVAILABLE is active*)								16#FF),
(*Transmission is VALID*)								USINT_TO_BYTE(REAL_TO_USINT((GVL.IOVD.P_X_T_Max_Wtr_BTMS_Heat.x))));
{endregion}

{region " SIGNAL AREA : NAME->P_X_T_Max_Wtr_BTMS_Cool LENGTH->8 STARTBIT :24"}
_FB_CanTx_Message_Unpack_415.X_Byte_3			:=
(*SELECT 1 : Is data valid and range is not exceed?*)	SEL((GVL.IOVD.P_X_T_Max_Wtr_BTMS_Cool.v AND NOT GVL.IOVD.P_X_T_Max_Wtr_BTMS_Cool.RangeExcd),
(*SELECT 2 : Is NOT AVAILABLE ?*)						SEL(GVL.IOVD.P_X_T_Max_Wtr_BTMS_Cool.na,
(*SELECT 3 : Is ERROR active ?*)						SEL(GVL.IOVD.P_X_T_Max_Wtr_BTMS_Cool.e,
(*DEFAULT VALUE assignment*)							0,
(*ERROR is active*)										16#FE),
(*NOT AVAILABLE is active*)								16#FF),
(*Transmission is VALID*)								USINT_TO_BYTE(REAL_TO_USINT((GVL.IOVD.P_X_T_Max_Wtr_BTMS_Cool.x))));
{endregion}

{region " SIGNAL AREA : NAME->P_X_T_Flr_Heat_Lim LENGTH->8 STARTBIT :32"}
_FB_CanTx_Message_Unpack_415.X_Byte_4			:=
(*SELECT 1 : Is data valid and range is not exceed?*)	SEL((GVL.IOVD.P_X_T_Flr_Heat_Lim.v AND NOT GVL.IOVD.P_X_T_Flr_Heat_Lim.RangeExcd),
(*SELECT 2 : Is NOT AVAILABLE ?*)						SEL(GVL.IOVD.P_X_T_Flr_Heat_Lim.na,
(*SELECT 3 : Is ERROR active ?*)						SEL(GVL.IOVD.P_X_T_Flr_Heat_Lim.e,
(*DEFAULT VALUE assignment*)							0,
(*ERROR is active*)										16#FE),
(*NOT AVAILABLE is active*)								16#FF),
(*Transmission is VALID*)								USINT_TO_BYTE(REAL_TO_USINT((GVL.IOVD.P_X_T_Flr_Heat_Lim.x))));
{endregion}

_FB_CanTx_Message_Unpack_415.X_Byte_5 				:= 16#FF;	
_FB_CanTx_Message_Unpack_415.X_Byte_6 				:= 16#FF;	
_FB_CanTx_Message_Unpack_415.X_Byte_7 				:= 16#FF;		
	
_FB_CanTx_Message_Unpack_415 (		C_Enable		:= GVL.IOVD.C_En_HVAC_Parameters_1_0X415,
     								Obj_CAN			:= ADR(GVL.IC.Obj_CAN0),
     								X_MsgID			:= 16#415,
     								Tm_CycleTime	:= TIME#500MS,							
     								N_Msg_Dlc		:= 8,
     								S_Extended		:= 0,
     								S_Sent_Ok   	=> GVL.IOVD.S_SentOk_HVAC_Parameters_1_0X415);	
{endregion}
//-----------------------------------------------------------------------------------------------------------------------------
//-----------------------------------------------------------------------------------------------------------------------------
{region " MESSAGE AREA :HVAC_Water_Temperature- ID:416"}

{region " SIGNAL AREA : NAME->X_T_BTMS_Wtr_Snsr_1 LENGTH->8 STARTBIT :0"}
_FB_CanTx_Message_Unpack_416.X_Byte_0					:=
(*SELECT 1 : Is data valid and range is not exceed?*)	SEL((GVL.IOVD.X_T_BTMS_Wtr_Snsr_1.v AND NOT GVL.IOVD.X_T_BTMS_Wtr_Snsr_1.RangeExcd),
(*SELECT 2 : Is NOT AVAILABLE ?*)						SEL(GVL.IOVD.X_T_BTMS_Wtr_Snsr_1.na,
(*SELECT 3 : Is ERROR active ?*)						SEL(GVL.IOVD.X_T_BTMS_Wtr_Snsr_1.e,
(*DEFAULT VALUE assignment*)							USINT_TO_BYTE(REAL_TO_USINT((0))),
(*ERROR is active*)										16#FE),
(*NOT AVAILABLE is active*)								16#FF),
(*Transmission is VALID*)								USINT_TO_BYTE(REAL_TO_USINT((GVL.IOVD.X_T_BTMS_Wtr_Snsr_1.x + 40))));
{endregion}

{region " SIGNAL AREA : NAME->X_T_BTMS_Wtr_Snsr_2 LENGTH->8 STARTBIT :8"}
_FB_CanTx_Message_Unpack_416.X_Byte_1					:=
(*SELECT 1 : Is data valid and range is not exceed?*)	SEL((GVL.IOVD.X_T_BTMS_Wtr_Snsr_2.v AND NOT GVL.IOVD.X_T_BTMS_Wtr_Snsr_2.RangeExcd),
(*SELECT 2 : Is NOT AVAILABLE ?*)						SEL(GVL.IOVD.X_T_BTMS_Wtr_Snsr_2.na,
(*SELECT 3 : Is ERROR active ?*)						SEL(GVL.IOVD.X_T_BTMS_Wtr_Snsr_2.e,
(*DEFAULT VALUE assignment*)							USINT_TO_BYTE(REAL_TO_USINT((0))),
(*ERROR is active*)										16#FE),
(*NOT AVAILABLE is active*)								16#FF),
(*Transmission is VALID*)								USINT_TO_BYTE(REAL_TO_USINT((GVL.IOVD.X_T_BTMS_Wtr_Snsr_2.x + 40))));
{endregion}

_FB_CanTx_Message_Unpack_416.X_Byte_2 				:= 16#FF;	
_FB_CanTx_Message_Unpack_416.X_Byte_3 				:= 16#FF;	
_FB_CanTx_Message_Unpack_416.X_Byte_4 				:= 16#FF;		
_FB_CanTx_Message_Unpack_416.X_Byte_5 				:= 16#FF;	
_FB_CanTx_Message_Unpack_416.X_Byte_6 				:= 16#FF;	
_FB_CanTx_Message_Unpack_416.X_Byte_7 				:= 16#FF;	
	
_FB_CanTx_Message_Unpack_416 (		C_Enable		:= GVL.IOVD.C_En_HVAC_Water_Temperature_0X416,
     								Obj_CAN			:= ADR(GVL.IC.Obj_CAN0),
     								X_MsgID			:= 16#416,
     								Tm_CycleTime	:= TIME#500MS,							
     								N_Msg_Dlc		:= 8,
     								S_Extended		:= 0,
     								S_Sent_Ok   	=> GVL.IOVD.S_SentOk_HVAC_Water_Temperature_0X416);	
{endregion}
//-----------------------------------------------------------------------------------------------------------------------------
//-----------------------------------------------------------------------------------------------------------------------------
{region " MESSAGE AREA :Arac_Menzil- ID:4C0"}

{region " SIGNAL AREA : NAME->X_Distn_Bat_Drvn LENGTH->16 STARTBIT :0"}
_FB_UNPACK_WORD_TO_BYTE_4 (
		X_WORD_0									:= 
(*SELECT 1 : Is data valid and range is not exceed?*)	SEL((GVL.IOVD.X_Distn_Bat_Drvn.v AND NOT GVL.IOVD.X_Distn_Bat_Drvn.RangeExcd),
(*SELECT 2 : Is NOT AVAILABLE ?*)						SEL(GVL.IOVD.X_Distn_Bat_Drvn.na,
(*SELECT 3 : Is ERROR active ?*)						SEL(GVL.IOVD.X_Distn_Bat_Drvn.e,
(*DEFAULT VALUE assignment*)							0,
(*ERROR is active*)										16#FEFE),
(*NOT AVAILABLE is active*)								16#FFFF),
(*Transmission is VALID*)								UINT_TO_WORD(REAL_TO_UINT((GVL.IOVD.X_Distn_Bat_Drvn.x)))),
		X_BYTE_0										=> _FB_CanTx_Message_4C0.X_Byte_0,
		X_BYTE_1										=> _FB_CanTx_Message_4C0.X_Byte_1);
{endregion}

{region " SIGNAL AREA : NAME->X_Distn_Rmn LENGTH->16 STARTBIT :16"}
_FB_UNPACK_WORD_TO_BYTE_5 (
		X_WORD_0									:= 
(*SELECT 1 : Is data valid and range is not exceed?*)	SEL((GVL.IOVD.X_Distn_Rmn.v AND NOT GVL.IOVD.X_Distn_Rmn.RangeExcd),
(*SELECT 2 : Is NOT AVAILABLE ?*)						SEL(GVL.IOVD.X_Distn_Rmn.na,
(*SELECT 3 : Is ERROR active ?*)						SEL(GVL.IOVD.X_Distn_Rmn.e,
(*DEFAULT VALUE assignment*)							0,
(*ERROR is active*)										16#FEFE),
(*NOT AVAILABLE is active*)								16#FFFF),
(*Transmission is VALID*)								UINT_TO_WORD(REAL_TO_UINT((GVL.IOVD.X_Distn_Rmn.x)))),
		X_BYTE_0										=> _FB_CanTx_Message_4C0.X_Byte_2,
		X_BYTE_1										=> _FB_CanTx_Message_4C0.X_Byte_3);
{endregion}

{region " SIGNAL AREA : NAME->X_Distn_Cat_Drvn LENGTH->32 STARTBIT :32"}
_FB_UNPACK_DWORD_TO_BYTE_0 (
		X_DWORD_0									:= 
(*SELECT 1 : Is data valid and range is not exceed?*)	SEL((GVL.IOVD.X_Distn_Cat_Drvn.v AND NOT GVL.IOVD.X_Distn_Cat_Drvn.RangeExcd),
(*SELECT 2 : Is NOT AVAILABLE ?*)						SEL(GVL.IOVD.X_Distn_Cat_Drvn.na,
(*SELECT 3 : Is ERROR active ?*)						SEL(GVL.IOVD.X_Distn_Cat_Drvn.e,
(*DEFAULT VALUE assignment*)							0,
(*ERROR is active*)										16#FEFEFEFE),
(*NOT AVAILABLE is active*)								16#FFFFFFFF),
(*Transmission is VALID*)								UDINT_TO_DWORD(REAL_TO_UDINT((GVL.IOVD.X_Distn_Cat_Drvn.x)))),
		X_BYTE_0										=> _FB_CanTx_Message_4C0.X_Byte_4,
		X_BYTE_1										=> _FB_CanTx_Message_4C0.X_Byte_5,
		X_BYTE_2										=> _FB_CanTx_Message_4C0.X_Byte_6,
		X_BYTE_3										=> _FB_CanTx_Message_4C0.X_Byte_7);
{endregion} 

_FB_CanTx_Message_4C0 (		C_Enable		:= GVL.IOVD.C_En_Arac_Menzil_0X4C0,
     						Obj_CAN			:= ADR(GVL.IC.Obj_CAN0),
     						X_MsgID			:= 16#4C0,
     						Tm_CycleTime	:= TIME#1000MS,
     						N_Msg_Dlc		:= 8,
     						S_Extended		:= 0,
     						S_Sent_Ok   	=> GVL.IOVD.S_SentOk_Arac_Menzil_0X4C0);
{endregion}
//-----------------------------------------------------------------------------------------------------------------------------
//-----------------------------------------------------------------------------------------------------------------------------
{region " MESSAGE AREA :Arac_Odometre- ID:4C1"}

{region " SIGNAL AREA : NAME->X_Om LENGTH->64 STARTBIT :0"}
_FB_UNPACK_DWORD_TO_BYTE_18 (
		X_DWORD_0									:= 
(*SELECT 1 : Is data valid and range is not exceed?*)	SEL((GVL.IOVD.X_Om.v AND NOT GVL.IOVD.X_Om.RangeExcd),
(*SELECT 2 : Is NOT AVAILABLE ?*)						SEL(GVL.IOVD.X_Om.na,
(*SELECT 3 : Is ERROR active ?*)						SEL(GVL.IOVD.X_Om.e,
(*DEFAULT VALUE assignment*)							0,
(*ERROR is active*)										16#FEFEFEFE),
(*NOT AVAILABLE is active*)								16#FFFFFFFF),
(*Transmission is VALID*)								UDINT_TO_DWORD(REAL_TO_UDINT((GVL.IOVD.X_Om.x)/0.1))),
		X_BYTE_0										=> _FB_CanTx_Message_4C1.X_Byte_0,
		X_BYTE_1										=> _FB_CanTx_Message_4C1.X_Byte_1,
		X_BYTE_2										=> _FB_CanTx_Message_4C1.X_Byte_2,
		X_BYTE_3										=> _FB_CanTx_Message_4C1.X_Byte_3);

_FB_CanTx_Message_4C1.X_Byte_4	:= 0;
_FB_CanTx_Message_4C1.X_Byte_5	:= 0;
_FB_CanTx_Message_4C1.X_Byte_6 	:= 0;
_FB_CanTx_Message_4C1.X_Byte_7	:= 0;				  
{endregion}

_FB_CanTx_Message_4C1 (		C_Enable		:= GVL.IOVD.C_En_Arac_Odometre_0X4C1,
     						Obj_CAN			:= ADR(GVL.IC.Obj_CAN0),
     						X_MsgID			:= 16#4C1,
     						Tm_CycleTime	:= TIME#1000MS,
     						N_Msg_Dlc		:= 8,
     						S_Extended		:= 0,
     						S_Sent_Ok   	=> GVL.IOVD.S_SentOk_Arac_Odometre_0X4C1);
{endregion}
//-----------------------------------------------------------------------------------------------------------------------------
//-----------------------------------------------------------------------------------------------------------------------------
{region " MESSAGE AREA :Arac_Surus_Enerji- ID:4C3"}

{region " SIGNAL AREA : NAME->X_E_Tr LENGTH->32 STARTBIT :0"}
_FB_UNPACK_DWORD_TO_BYTE_1 (
		X_DWORD_0									:= 
(*SELECT 1 : Is data valid and range is not exceed?*)	SEL((GVL.IOVD.X_E_Tr.v AND NOT GVL.IOVD.X_E_Tr.RangeExcd),
(*SELECT 2 : Is NOT AVAILABLE ?*)						SEL(GVL.IOVD.X_E_Tr.na,
(*SELECT 3 : Is ERROR active ?*)						SEL(GVL.IOVD.X_E_Tr.e,
(*DEFAULT VALUE assignment*)							0,
(*ERROR is active*)										16#FEFEFEFE),
(*NOT AVAILABLE is active*)								16#FFFFFFFF),
(*Transmission is VALID*)								UDINT_TO_DWORD(REAL_TO_UDINT((GVL.IOVD.X_E_Tr.x)/0.1))),
		X_BYTE_0										=> _FB_CanTx_Message_4C3.X_Byte_0,
		X_BYTE_1										=> _FB_CanTx_Message_4C3.X_Byte_1,
		X_BYTE_2										=> _FB_CanTx_Message_4C3.X_Byte_2,
		X_BYTE_3										=> _FB_CanTx_Message_4C3.X_Byte_3);
{endregion}

{region " SIGNAL AREA : NAME->X_E_Regn LENGTH->32 STARTBIT :32"}
_FB_UNPACK_DWORD_TO_BYTE_2 (
		X_DWORD_0									:= 
(*SELECT 1 : Is data valid and range is not exceed?*)	SEL((GVL.IOVD.X_E_Regn.v AND NOT GVL.IOVD.X_E_Regn.RangeExcd),
(*SELECT 2 : Is NOT AVAILABLE ?*)						SEL(GVL.IOVD.X_E_Regn.na,
(*SELECT 3 : Is ERROR active ?*)						SEL(GVL.IOVD.X_E_Regn.e,
(*DEFAULT VALUE assignment*)							0,
(*ERROR is active*)										16#FEFEFEFE),
(*NOT AVAILABLE is active*)								16#FFFFFFFF),
(*Transmission is VALID*)								UDINT_TO_DWORD(REAL_TO_UDINT((GVL.IOVD.X_E_Regn.x)/0.1))),
		X_BYTE_0										=> _FB_CanTx_Message_4C3.X_Byte_4,
		X_BYTE_1										=> _FB_CanTx_Message_4C3.X_Byte_5,
		X_BYTE_2										=> _FB_CanTx_Message_4C3.X_Byte_6,
		X_BYTE_3										=> _FB_CanTx_Message_4C3.X_Byte_7);
{endregion}

_FB_CanTx_Message_4C3 (		C_Enable		:= GVL.IOVD.C_En_Arac_Surus_Enerji_0X4C3,
     						Obj_CAN			:= ADR(GVL.IC.Obj_CAN0),
     						X_MsgID			:= 16#4C3,
     						Tm_CycleTime	:= TIME#1000MS,
     						N_Msg_Dlc		:= 8,
     						S_Extended		:= 0,
     						S_Sent_Ok   	=> GVL.IOVD.S_SentOk_Arac_Surus_Enerji_0X4C3);
{endregion}
//-----------------------------------------------------------------------------------------------------------------------------
//-----------------------------------------------------------------------------------------------------------------------------
{region " MESSAGE AREA :Arac_Tuketilen_Enerji_1- ID:4C4"}

{region " SIGNAL AREA : NAME->X_E_Aux_DC LENGTH->32 STARTBIT :0"}
_FB_UNPACK_DWORD_TO_BYTE_3 (
		X_DWORD_0									:= 
(*SELECT 1 : Is data valid and range is not exceed?*)	SEL((GVL.IOVD.X_E_Aux_DC.v AND NOT GVL.IOVD.X_E_Aux_DC.RangeExcd),
(*SELECT 2 : Is NOT AVAILABLE ?*)						SEL(GVL.IOVD.X_E_Aux_DC.na,
(*SELECT 3 : Is ERROR active ?*)						SEL(GVL.IOVD.X_E_Aux_DC.e,
(*DEFAULT VALUE assignment*)							0,
(*ERROR is active*)										16#FEFEFEFE),
(*NOT AVAILABLE is active*)								16#FFFFFFFF),
(*Transmission is VALID*)								UDINT_TO_DWORD(REAL_TO_UDINT((GVL.IOVD.X_E_Aux_DC.x)/0.1))),
		X_BYTE_0										=> _FB_CanTx_Message_4C4.X_Byte_0,
		X_BYTE_1										=> _FB_CanTx_Message_4C4.X_Byte_1,
		X_BYTE_2										=> _FB_CanTx_Message_4C4.X_Byte_2,
		X_BYTE_3										=> _FB_CanTx_Message_4C4.X_Byte_3);
{endregion}

{region " SIGNAL AREA : NAME->X_E_Aux_DC_24V LENGTH->32 STARTBIT :32"}
_FB_UNPACK_DWORD_TO_BYTE_4 (
		X_DWORD_0									:= 
(*SELECT 1 : Is data valid and range is not exceed?*)	SEL((GVL.IOVD.X_E_Aux_DC_24V.v AND NOT GVL.IOVD.X_E_Aux_DC_24V.RangeExcd),
(*SELECT 2 : Is NOT AVAILABLE ?*)						SEL(GVL.IOVD.X_E_Aux_DC_24V.na,
(*SELECT 3 : Is ERROR active ?*)						SEL(GVL.IOVD.X_E_Aux_DC_24V.e,
(*DEFAULT VALUE assignment*)							0,
(*ERROR is active*)										16#FEFEFEFE),
(*NOT AVAILABLE is active*)								16#FFFFFFFF),
(*Transmission is VALID*)								UDINT_TO_DWORD(REAL_TO_UDINT((GVL.IOVD.X_E_Aux_DC_24V.x)/0.1))),
		X_BYTE_0										=> _FB_CanTx_Message_4C4.X_Byte_4,
		X_BYTE_1										=> _FB_CanTx_Message_4C4.X_Byte_5,
		X_BYTE_2										=> _FB_CanTx_Message_4C4.X_Byte_6,
		X_BYTE_3										=> _FB_CanTx_Message_4C4.X_Byte_7);
{endregion}

_FB_CanTx_Message_4C4 (		C_Enable		:= GVL.IOVD.C_En_Arac_Tuketilen_Enerji_1_0X4C4,
     						Obj_CAN			:= ADR(GVL.IC.Obj_CAN0),
     						X_MsgID			:= 16#4C4,
     						Tm_CycleTime	:= TIME#1000MS,
     						N_Msg_Dlc		:= 8,
     						S_Extended		:= 0,
     						S_Sent_Ok   	=> GVL.IOVD.S_SentOk_Arac_Tuketilen_Enerji_1_0X4C4);
{endregion}
//-----------------------------------------------------------------------------------------------------------------------------
//-----------------------------------------------------------------------------------------------------------------------------
{region " MESSAGE AREA :Arac_Tuketilen_Enerji_2- ID:4C5"}

{region " SIGNAL AREA : NAME->X_E_Aux_AC LENGTH->32 STARTBIT :0"}
_FB_UNPACK_DWORD_TO_BYTE_5 (
		X_DWORD_0									:= 
(*SELECT 1 : Is data valid and range is not exceed?*)	SEL((GVL.IOVD.X_E_Aux_AC.v AND NOT GVL.IOVD.X_E_Aux_AC.RangeExcd),
(*SELECT 2 : Is NOT AVAILABLE ?*)						SEL(GVL.IOVD.X_E_Aux_AC.na,
(*SELECT 3 : Is ERROR active ?*)						SEL(GVL.IOVD.X_E_Aux_AC.e,
(*DEFAULT VALUE assignment*)							0,
(*ERROR is active*)										16#FEFEFEFE),
(*NOT AVAILABLE is active*)								16#FFFFFFFF),
(*Transmission is VALID*)								UDINT_TO_DWORD(REAL_TO_UDINT((GVL.IOVD.X_E_Aux_AC.x)/0.1))),
		X_BYTE_0										=> _FB_CanTx_Message_4C5.X_Byte_0,
		X_BYTE_1										=> _FB_CanTx_Message_4C5.X_Byte_1,
		X_BYTE_2										=> _FB_CanTx_Message_4C5.X_Byte_2,
		X_BYTE_3										=> _FB_CanTx_Message_4C5.X_Byte_3);
{endregion}

{region " SIGNAL AREA : NAME->X_E_Cosu LENGTH->32 STARTBIT :32"}
_FB_UNPACK_DWORD_TO_BYTE_6 (
		X_DWORD_0									:= 
(*SELECT 1 : Is data valid and range is not exceed?*)	SEL((GVL.IOVD.X_E_Cosu.v AND NOT GVL.IOVD.X_E_Cosu.RangeExcd),
(*SELECT 2 : Is NOT AVAILABLE ?*)						SEL(GVL.IOVD.X_E_Cosu.na,
(*SELECT 3 : Is ERROR active ?*)						SEL(GVL.IOVD.X_E_Cosu.e,
(*DEFAULT VALUE assignment*)							0,
(*ERROR is active*)										16#FEFEFEFE),
(*NOT AVAILABLE is active*)								16#FFFFFFFF),
(*Transmission is VALID*)								UDINT_TO_DWORD(REAL_TO_UDINT((GVL.IOVD.X_E_Cosu.x)/0.1))),
		X_BYTE_0										=> _FB_CanTx_Message_4C5.X_Byte_4,
		X_BYTE_1										=> _FB_CanTx_Message_4C5.X_Byte_5,
		X_BYTE_2										=> _FB_CanTx_Message_4C5.X_Byte_6,
		X_BYTE_3										=> _FB_CanTx_Message_4C5.X_Byte_7);
{endregion}

_FB_CanTx_Message_4C5 (		C_Enable		:= GVL.IOVD.C_En_Arac_Tuketilen_Enerji_2_0X4C5,
     						Obj_CAN			:= ADR(GVL.IC.Obj_CAN0),
     						X_MsgID			:= 16#4C5,
     						Tm_CycleTime	:= TIME#1000MS,
     						N_Msg_Dlc		:= 8,
     						S_Extended		:= 0,
     						S_Sent_Ok   	=> GVL.IOVD.S_SentOk_Arac_Tuketilen_Enerji_2_0X4C5);
{endregion}
//-----------------------------------------------------------------------------------------------------------------------------
//-----------------------------------------------------------------------------------------------------------------------------
{region " MESSAGE AREA :Arac_Kapasite- ID:4C6"}

{region " SIGNAL AREA : NAME->X_Capcty_Act LENGTH->32 STARTBIT :0"}
_FB_UNPACK_DWORD_TO_BYTE_7 (
		X_DWORD_0									:= 
(*SELECT 1 : Is data valid and range is not exceed?*)	SEL((GVL.IOVD.X_Capcty_Act.v AND NOT GVL.IOVD.X_Capcty_Act.RangeExcd),
(*SELECT 2 : Is NOT AVAILABLE ?*)						SEL(GVL.IOVD.X_Capcty_Act.na,
(*SELECT 3 : Is ERROR active ?*)						SEL(GVL.IOVD.X_Capcty_Act.e,
(*DEFAULT VALUE assignment*)							0,
(*ERROR is active*)										16#FEFEFEFE),
(*NOT AVAILABLE is active*)								16#FFFFFFFF),
(*Transmission is VALID*)								UDINT_TO_DWORD(REAL_TO_UDINT((GVL.IOVD.X_Capcty_Act.x)/0.1))),
		X_BYTE_0										=> _FB_CanTx_Message_4C6.X_Byte_0,
		X_BYTE_1										=> _FB_CanTx_Message_4C6.X_Byte_1,
		X_BYTE_2										=> _FB_CanTx_Message_4C6.X_Byte_2,
		X_BYTE_3										=> _FB_CanTx_Message_4C6.X_Byte_3);
{endregion}

{region " SIGNAL AREA : NAME->X_Capcty_Rmn LENGTH->32 STARTBIT :32"}
_FB_UNPACK_DWORD_TO_BYTE_8 (
		X_DWORD_0									:= 
(*SELECT 1 : Is data valid and range is not exceed?*)	SEL((GVL.IOVD.X_Capcty_Rmn.v AND NOT GVL.IOVD.X_Capcty_Rmn.RangeExcd),
(*SELECT 2 : Is NOT AVAILABLE ?*)						SEL(GVL.IOVD.X_Capcty_Rmn.na,
(*SELECT 3 : Is ERROR active ?*)						SEL(GVL.IOVD.X_Capcty_Rmn.e,
(*DEFAULT VALUE assignment*)							0,
(*ERROR is active*)										16#FEFEFEFE),
(*NOT AVAILABLE is active*)								16#FFFFFFFF),
(*Transmission is VALID*)								UDINT_TO_DWORD(REAL_TO_UDINT((GVL.IOVD.X_Capcty_Rmn.x)/0.1))),
		X_BYTE_0										=> _FB_CanTx_Message_4C6.X_Byte_4,
		X_BYTE_1										=> _FB_CanTx_Message_4C6.X_Byte_5,
		X_BYTE_2										=> _FB_CanTx_Message_4C6.X_Byte_6,
		X_BYTE_3										=> _FB_CanTx_Message_4C6.X_Byte_7);
{endregion}

_FB_CanTx_Message_4C6 (		C_Enable		:= GVL.IOVD.C_En_Arac_Kapasite_0X4C6,
     						Obj_CAN			:= ADR(GVL.IC.Obj_CAN0),
     						X_MsgID			:= 16#4C6,
     						Tm_CycleTime	:= TIME#1000ms,
     						N_Msg_Dlc		:= 8,
     						S_Extended		:= 0,
     						S_Sent_Ok  		=> GVL.IOVD.S_SentOk_Arac_Kapasite_0X4C6);
{endregion}
//-----------------------------------------------------------------------------------------------------------------------------
//-----------------------------------------------------------------------------------------------------------------------------
{region " MESSAGE AREA :Arac_Sureler- ID:4C7"}

{region " SIGNAL AREA : NAME->X_Tm_Bat_Drvn LENGTH->16 STARTBIT :0"}
_FB_UNPACK_WORD_TO_BYTE_6 (
		X_WORD_0									:= 
(*SELECT 1 : Is data valid and range is not exceed?*)	SEL((GVL.IOVD.X_Tm_Bat_Drvn.v AND NOT GVL.IOVD.X_Tm_Bat_Drvn.RangeExcd),
(*SELECT 2 : Is NOT AVAILABLE ?*)						SEL(GVL.IOVD.X_Tm_Bat_Drvn.na,
(*SELECT 3 : Is ERROR active ?*)						SEL(GVL.IOVD.X_Tm_Bat_Drvn.e,
(*DEFAULT VALUE assignment*)							0,
(*ERROR is active*)										16#FEFE),
(*NOT AVAILABLE is active*)								16#FFFF),
(*Transmission is VALID*)								UINT_TO_WORD(REAL_TO_UINT((GVL.IOVD.X_Tm_Bat_Drvn.x)))),
		X_BYTE_0										=> _FB_CanTx_Message_4C7.X_Byte_0,
		X_BYTE_1										=> _FB_CanTx_Message_4C7.X_Byte_1);
{endregion}

{region " SIGNAL AREA : NAME->X_Tm_Cat_Drvn LENGTH->16 STARTBIT :16"}
_FB_UNPACK_WORD_TO_BYTE_7 (
		X_WORD_0									:= 
(*SELECT 1 : Is data valid and range is not exceed?*)	SEL((GVL.IOVD.X_Tm_Cat_Drvn.v AND NOT GVL.IOVD.X_Tm_Cat_Drvn.RangeExcd),
(*SELECT 2 : Is NOT AVAILABLE ?*)						SEL(GVL.IOVD.X_Tm_Cat_Drvn.na,
(*SELECT 3 : Is ERROR active ?*)						SEL(GVL.IOVD.X_Tm_Cat_Drvn.e,
(*DEFAULT VALUE assignment*)							0,
(*ERROR is active*)										16#FEFE),
(*NOT AVAILABLE is active*)								16#FFFF),
(*Transmission is VALID*)								UINT_TO_WORD(REAL_TO_UINT((GVL.IOVD.X_Tm_Cat_Drvn.x)))),
		X_BYTE_0										=> _FB_CanTx_Message_4C7.X_Byte_2,
		X_BYTE_1										=> _FB_CanTx_Message_4C7.X_Byte_3);
{endregion}

{region " SIGNAL AREA : NAME->X_Tm_Wt LENGTH->16 STARTBIT :32"}
_FB_UNPACK_WORD_TO_BYTE_8 (
		X_WORD_0									:= 
(*SELECT 1 : Is data valid and range is not exceed?*)	SEL((GVL.IOVD.X_Tm_Wt.v AND NOT GVL.IOVD.X_Tm_Wt.RangeExcd),
(*SELECT 2 : Is NOT AVAILABLE ?*)						SEL(GVL.IOVD.X_Tm_Wt.na,
(*SELECT 3 : Is ERROR active ?*)						SEL(GVL.IOVD.X_Tm_Wt.e,
(*DEFAULT VALUE assignment*)							0,
(*ERROR is active*)										16#FEFE),
(*NOT AVAILABLE is active*)								16#FFFF),
(*Transmission is VALID*)								UINT_TO_WORD(REAL_TO_UINT((GVL.IOVD.X_Tm_Wt.x)))),
		X_BYTE_0										=> _FB_CanTx_Message_4C7.X_Byte_4,
		X_BYTE_1										=> _FB_CanTx_Message_4C7.X_Byte_5);
{endregion}

{region " SIGNAL AREA : NAME->X_Tm_HVAC_On LENGTH->16 STARTBIT :48"}
_FB_UNPACK_WORD_TO_BYTE_9 (
		X_WORD_0									:= 
(*SELECT 1 : Is data valid and range is not exceed?*)	SEL((GVL.IOVD.X_Tm_HVAC_On.v AND NOT GVL.IOVD.X_Tm_HVAC_On.RangeExcd),
(*SELECT 2 : Is NOT AVAILABLE ?*)						SEL(GVL.IOVD.X_Tm_HVAC_On.na,
(*SELECT 3 : Is ERROR active ?*)						SEL(GVL.IOVD.X_Tm_HVAC_On.e,
(*DEFAULT VALUE assignment*)							0,
(*ERROR is active*)										16#FEFE),
(*NOT AVAILABLE is active*)								16#FFFF),
(*Transmission is VALID*)								UINT_TO_WORD(REAL_TO_UINT((GVL.IOVD.X_Tm_HVAC_On.x)))),
		X_BYTE_0										=> _FB_CanTx_Message_4C7.X_Byte_6,
		X_BYTE_1										=> _FB_CanTx_Message_4C7.X_Byte_7);
{endregion}

_FB_CanTx_Message_4C7 (		C_Enable		:= GVL.IOVD.C_En_Arac_Sureler_0X4C7,
     						Obj_CAN			:= ADR(GVL.IC.Obj_CAN0),
     						X_MsgID			:= 16#4C7,
     						Tm_CycleTime	:= TIME#1000MS,
     						N_Msg_Dlc		:= 8,
     						S_Extended		:= 0,
     						S_Sent_Ok   	=> GVL.IOVD.S_SentOk_Arac_Sureler_0X4C7);
{endregion}
//-----------------------------------------------------------------------------------------------------------------------------
//-----------------------------------------------------------------------------------------------------------------------------
{region " MESSAGE AREA :Arac_Toplam_Tuketilen_Enerji- ID:4C8"}

{region " SIGNAL AREA : NAME->X_E_Tot_Cosu LENGTH->32 STARTBIT :0"}
_FB_UNPACK_DWORD_TO_BYTE_9 (
		X_DWORD_0									:= 
(*SELECT 1 : Is data valid and range is not exceed?*)	SEL((GVL.IOVD.X_E_Tot_Cosu.v AND NOT GVL.IOVD.X_E_Tot_Cosu.RangeExcd),
(*SELECT 2 : Is NOT AVAILABLE ?*)						SEL(GVL.IOVD.X_E_Tot_Cosu.na,
(*SELECT 3 : Is ERROR active ?*)						SEL(GVL.IOVD.X_E_Tot_Cosu.e,
(*DEFAULT VALUE assignment*)							0,
(*ERROR is active*)										16#FEFEFEFE),
(*NOT AVAILABLE is active*)								16#FFFFFFFF),
(*Transmission is VALID*)								UDINT_TO_DWORD(REAL_TO_UDINT((GVL.IOVD.X_E_Tot_Cosu.x)/0.1))),
		X_BYTE_0										=> _FB_CanTx_Message_4C8.X_Byte_0,
		X_BYTE_1										=> _FB_CanTx_Message_4C8.X_Byte_1,
		X_BYTE_2										=> _FB_CanTx_Message_4C8.X_Byte_2,
		X_BYTE_3										=> _FB_CanTx_Message_4C8.X_Byte_3);
{endregion}

{region " SIGNAL AREA : NAME->X_Avg_Cosu_Opp LENGTH->16 STARTBIT :32"}
_FB_UNPACK_WORD_TO_BYTE_12 (
		X_WORD_0									:= 
(*SELECT 1 : Is data valid and range is not exceed?*)	SEL((GVL.IOVD.X_Avg_Cosu_Opp.v AND NOT GVL.IOVD.X_Avg_Cosu_Opp.RangeExcd),
(*SELECT 2 : Is NOT AVAILABLE ?*)						SEL(GVL.IOVD.X_Avg_Cosu_Opp.na,
(*SELECT 3 : Is ERROR active ?*)						SEL(GVL.IOVD.X_Avg_Cosu_Opp.e,
(*DEFAULT VALUE assignment*)							0,
(*ERROR is active*)										16#FEFE),
(*NOT AVAILABLE is active*)								16#FFFF),
(*Transmission is VALID*)								UINT_TO_WORD(REAL_TO_UINT((GVL.IOVD.X_Avg_Cosu_Opp.x)/0.001))),
		X_BYTE_0										=> _FB_CanTx_Message_4C8.X_Byte_4,
		X_BYTE_1										=> _FB_CanTx_Message_4C8.X_Byte_5);
{endregion}
		
_FB_CanTx_Message_4C8.X_Byte_6 		:= 16#FF;
_FB_CanTx_Message_4C8.X_Byte_7 		:= 16#FF;
_FB_CanTx_Message_4C8 (		C_Enable		:= GVL.IOVD.C_En_Arac_Toplam_Tuketilen_Enerji_0X4C8,
     						Obj_CAN			:= ADR(GVL.IC.Obj_CAN0),
     						X_MsgID			:= 16#4C8,
     						Tm_CycleTime	:= TIME#1000MS,
     						N_Msg_Dlc		:= 8,
     						S_Extended		:= 0,
     						S_Sent_Ok   	=> GVL.IOVD.S_SentOk_Arac_Toplam_Tuketilen_Enerji_0X4C8);
{endregion}
//-----------------------------------------------------------------------------------------------------------------------------
//-----------------------------------------------------------------------------------------------------------------------------
{region " MESSAGE AREA :Arac_Genel_Istatistik_2- ID:4C9"}

{region " SIGNAL AREA : NAME->X_Daily_Avg_Cosu LENGTH->16 STARTBIT :0"}
_FB_UNPACK_WORD_TO_BYTE_10 (
		X_WORD_0									:= 
(*SELECT 1 : Is data valid and range is not exceed?*)	SEL((GVL.IOVD.X_Daily_Avg_Cosu.v AND NOT GVL.IOVD.X_Daily_Avg_Cosu.RangeExcd),
(*SELECT 2 : Is NOT AVAILABLE ?*)						SEL(GVL.IOVD.X_Daily_Avg_Cosu.na,
(*SELECT 3 : Is ERROR active ?*)						SEL(GVL.IOVD.X_Daily_Avg_Cosu.e,
(*DEFAULT VALUE assignment*)							0,
(*ERROR is active*)										16#FEFE),
(*NOT AVAILABLE is active*)								16#FFFF),
(*Transmission is VALID*)								UINT_TO_WORD(REAL_TO_UINT((GVL.IOVD.X_Daily_Avg_Cosu.x)/0.001))),
		X_BYTE_0										=> _FB_CanTx_Message_4C9.X_Byte_0,
		X_BYTE_1										=> _FB_CanTx_Message_4C9.X_Byte_1);
{endregion}

{region " SIGNAL AREA : NAME->X_Trp_Distn LENGTH->32 STARTBIT :16"}
_FB_UNPACK_DWORD_TO_BYTE_10 (
		X_DWORD_0									:= 
(*SELECT 1 : Is data valid and range is not exceed?*)	SEL((GVL.IOVD.X_Trp_Distn.v AND NOT GVL.IOVD.X_Trp_Distn.RangeExcd),
(*SELECT 2 : Is NOT AVAILABLE ?*)						SEL(GVL.IOVD.X_Trp_Distn.na,
(*SELECT 3 : Is ERROR active ?*)						SEL(GVL.IOVD.X_Trp_Distn.e,
(*DEFAULT VALUE assignment*)							0,
(*ERROR is active*)										16#FEFEFEFE),
(*NOT AVAILABLE is active*)								16#FFFFFFFF),
(*Transmission is VALID*)								UDINT_TO_DWORD(REAL_TO_UDINT((GVL.IOVD.X_Trp_Distn.x)/0.1))),
		X_BYTE_0										=> _FB_CanTx_Message_4C9.X_Byte_2,
		X_BYTE_1										=> _FB_CanTx_Message_4C9.X_Byte_3,
		X_BYTE_2										=> _FB_CanTx_Message_4C9.X_Byte_4,
		X_BYTE_3										=> _FB_CanTx_Message_4C9.X_Byte_5);
{endregion}

{region " SIGNAL AREA : NAME->X_U_ECU_Sp LENGTH->16 STARTBIT :48"}
_FB_UNPACK_WORD_TO_BYTE_14(
		X_WORD_0									:= 
(*SELECT 1 : Is data valid and range is not exceed?*)	SEL((GVL.IOVD.X_U_ECU_Sp.v AND NOT GVL.IOVD.X_U_ECU_Sp.RangeExcd),
(*SELECT 2 : Is NOT AVAILABLE ?*)						SEL(GVL.IOVD.X_U_ECU_Sp.na,
(*SELECT 3 : Is ERROR active ?*)						SEL(GVL.IOVD.X_U_ECU_Sp.e,
(*DEFAULT VALUE assignment*)							0,
(*ERROR is active*)										16#FEFE),
(*NOT AVAILABLE is active*)								16#FFFF),
(*Transmission is VALID*)								UINT_TO_WORD(REAL_TO_UINT((GVL.IOVD.X_U_ECU_Sp.x)))),
		X_BYTE_0=> _FB_CanTx_Message_4C9.X_Byte_6,
		X_BYTE_1=> _FB_CanTx_Message_4C9.X_Byte_7);
{endregion}	

_FB_CanTx_Message_4C9 (		C_Enable		:= GVL.IOVD.C_En_Arac_Genel_Istatistik_2_0X4C9,
     						Obj_CAN			:= ADR(GVL.IC.Obj_CAN0),
     						X_MsgID			:= 16#4C9,
     						Tm_CycleTime	:= TIME#1000MS,
     						N_Msg_Dlc		:= 8,
     						S_Extended		:= 0,
     						S_Sent_Ok   	=> GVL.IOVD.S_SentOk_Arac_Genel_Istatistik_2_0X4C9);
{endregion}
//-----------------------------------------------------------------------------------------------------------------------------
//-----------------------------------------------------------------------------------------------------------------------------
{region " MESSAGE AREA :Klima_Calisma_Sureleri_1- ID:4CA"}

{region " SIGNAL AREA : NAME->N_Hvac_Drv_Op_Cnt LENGTH->32 STARTBIT :0"}
_FB_UNPACK_DWORD_TO_BYTE_11 (
		X_DWORD_0									:= 
(*SELECT 1 : Is data valid and range is not exceed?*)	SEL((GVL.IOVD.N_Hvac_Drv_Op_Cnt.v AND NOT GVL.IOVD.N_Hvac_Drv_Op_Cnt.RangeExcd),
(*SELECT 2 : Is NOT AVAILABLE ?*)						SEL(GVL.IOVD.N_Hvac_Drv_Op_Cnt.na,
(*SELECT 3 : Is ERROR active ?*)						SEL(GVL.IOVD.N_Hvac_Drv_Op_Cnt.e,
(*DEFAULT VALUE assignment*)							0,
(*ERROR is active*)										16#FEFEFEFE),
(*NOT AVAILABLE is active*)								16#FFFFFFFF),
(*Transmission is VALID*)								UDINT_TO_DWORD(GVL.IOVD.N_Hvac_Drv_Op_Cnt.x)),
		X_BYTE_0										=> _FB_CanTx_Message_4CA.X_Byte_0,
		X_BYTE_1										=> _FB_CanTx_Message_4CA.X_Byte_1,
		X_BYTE_2										=> _FB_CanTx_Message_4CA.X_Byte_2,
		X_BYTE_3										=> _FB_CanTx_Message_4CA.X_Byte_3);
{endregion}

{region " SIGNAL AREA : NAME->N_Hvac_Pass1_Op_Cnt LENGTH->32 STARTBIT :32"}
_FB_UNPACK_DWORD_TO_BYTE_12 (
		X_DWORD_0									:= 
(*SELECT 1 : Is data valid and range is not exceed?*)	SEL((GVL.IOVD.N_Hvac_Pass1_Op_Cnt.v AND NOT GVL.IOVD.N_Hvac_Pass1_Op_Cnt.RangeExcd),
(*SELECT 2 : Is NOT AVAILABLE ?*)						SEL(GVL.IOVD.N_Hvac_Pass1_Op_Cnt.na,
(*SELECT 3 : Is ERROR active ?*)						SEL(GVL.IOVD.N_Hvac_Pass1_Op_Cnt.e,
(*DEFAULT VALUE assignment*)							0,
(*ERROR is active*)										16#FEFEFEFE),
(*NOT AVAILABLE is active*)								16#FFFFFFFF),
(*Transmission is VALID*)								UDINT_TO_DWORD(GVL.IOVD.N_Hvac_Pass1_Op_Cnt.x)),
		X_BYTE_0										=> _FB_CanTx_Message_4CA.X_Byte_4,
		X_BYTE_1										=> _FB_CanTx_Message_4CA.X_Byte_5,
		X_BYTE_2										=> _FB_CanTx_Message_4CA.X_Byte_6,
		X_BYTE_3										=> _FB_CanTx_Message_4CA.X_Byte_7);
{endregion}

_FB_CanTx_Message_4CA (		C_Enable		:= GVL.IOVD.C_En_Klima_Calisma_Sureleri_1_0X4CA,
     						Obj_CAN			:= ADR(GVL.IC.Obj_CAN0),
     						X_MsgID			:= 16#4CA,
     						Tm_CycleTime	:= TIME#1000MS,
     						N_Msg_Dlc		:= 8,
     						S_Extended		:= 0,
     						S_Sent_Ok   	=> GVL.IOVD.S_SentOk_Klima_Calisma_Sureleri_1_0X4CA);
{endregion}
//-----------------------------------------------------------------------------------------------------------------------------
//-----------------------------------------------------------------------------------------------------------------------------
{region " MESSAGE AREA :Klima_Calisma_Sureleri_2- ID:4CB"}

{region " SIGNAL AREA : NAME->N_Hvac_Pass2_Op_Cnt LENGTH->32 STARTBIT :0"}
_FB_UNPACK_DWORD_TO_BYTE_13 (
		X_DWORD_0									:= 
(*SELECT 1 : Is data valid and range is not exceed?*)	SEL((GVL.IOVD.N_Hvac_Pass2_Op_Cnt.v AND NOT GVL.IOVD.N_Hvac_Pass2_Op_Cnt.RangeExcd),
(*SELECT 2 : Is NOT AVAILABLE ?*)						SEL(GVL.IOVD.N_Hvac_Pass2_Op_Cnt.na,
(*SELECT 3 : Is ERROR active ?*)						SEL(GVL.IOVD.N_Hvac_Pass2_Op_Cnt.e,
(*DEFAULT VALUE assignment*)							0,
(*ERROR is active*)										16#FEFEFEFE),
(*NOT AVAILABLE is active*)								16#FFFFFFFF),
(*Transmission is VALID*)								UDINT_TO_DWORD(GVL.IOVD.N_Hvac_Pass2_Op_Cnt.x)),
		X_BYTE_0										=> _FB_CanTx_Message_4CB.X_Byte_0,
		X_BYTE_1										=> _FB_CanTx_Message_4CB.X_Byte_1,
		X_BYTE_2										=> _FB_CanTx_Message_4CB.X_Byte_2,
		X_BYTE_3										=> _FB_CanTx_Message_4CB.X_Byte_3);
{endregion}

{region " SIGNAL AREA : NAME->N_Btms_Op_Cnt LENGTH->32 STARTBIT :32"}
_FB_UNPACK_DWORD_TO_BYTE_14 (
		X_DWORD_0									:= 
(*SELECT 1 : Is data valid and range is not exceed?*)	SEL((GVL.IOVD.N_Btms_Op_Cnt.v AND NOT GVL.IOVD.N_Btms_Op_Cnt.RangeExcd),
(*SELECT 2 : Is NOT AVAILABLE ?*)						SEL(GVL.IOVD.N_Btms_Op_Cnt.na,
(*SELECT 3 : Is ERROR active ?*)						SEL(GVL.IOVD.N_Btms_Op_Cnt.e,
(*DEFAULT VALUE assignment*)							0,
(*ERROR is active*)										16#FEFEFEFE),
(*NOT AVAILABLE is active*)								16#FFFFFFFF),
(*Transmission is VALID*)								UDINT_TO_DWORD(GVL.IOVD.N_Btms_Op_Cnt.x)),
		X_BYTE_0										=> _FB_CanTx_Message_4CB.X_Byte_4,
		X_BYTE_1										=> _FB_CanTx_Message_4CB.X_Byte_5,
		X_BYTE_2										=> _FB_CanTx_Message_4CB.X_Byte_6,
		X_BYTE_3										=> _FB_CanTx_Message_4CB.X_Byte_7);
{endregion}

_FB_CanTx_Message_4CB (		C_Enable		:= GVL.IOVD.C_En_Klima_Calisma_Sureleri_2_0X4CB,
     						Obj_CAN			:= ADR(GVL.IC.Obj_CAN0),
     						X_MsgID			:= 16#4CB,
     						Tm_CycleTime	:= TIME#1000MS,
     						N_Msg_Dlc		:= 8,
     						S_Extended		:= 0,
     						S_Sent_Ok   	=> GVL.IOVD.S_SentOk_Klima_Calisma_Sureleri_2_0X4CB);
{endregion}
//-----------------------------------------------------------------------------------------------------------------------------
//-----------------------------------------------------------------------------------------------------------------------------
{region " MESSAGE AREA :Sayicilar_1- ID:4CC"}

// PR1006_REV_002519_TIMTRO
{region " SIGNAL AREA : NAME->N_Bat_Cycle_Cnt LENGTH->32 STARTBIT :0"}
_FB_UNPACK_DWORD_TO_BYTE_15 (
		X_DWORD_0									:= 
(*SELECT 1 : Is data valid and range is not exceed?*)	SEL((GVL.IOVD.N_Air_Cmp_Op_Cnt.v AND NOT GVL.IOVD.N_Air_Cmp_Op_Cnt.RangeExcd),
(*SELECT 2 : Is NOT AVAILABLE ?*)						SEL(GVL.IOVD.N_Air_Cmp_Op_Cnt.na,
(*SELECT 3 : Is ERROR active ?*)						SEL(GVL.IOVD.N_Air_Cmp_Op_Cnt.e,
(*DEFAULT VALUE assignment*)							0,
(*ERROR is active*)										16#FEFEFEFE),
(*NOT AVAILABLE is active*)								16#FFFFFFFF),
(*Transmission is VALID*)								UDINT_TO_DWORD(GVL.IOVD.N_Air_Cmp_Op_Cnt.x)),
		X_BYTE_0										=> _FB_CanTx_Message_Unpack_4CC.X_Byte_0,
		X_BYTE_1										=> _FB_CanTx_Message_Unpack_4CC.X_Byte_1,
		X_BYTE_2										=> _FB_CanTx_Message_Unpack_4CC.X_Byte_2,
		X_BYTE_3										=> _FB_CanTx_Message_Unpack_4CC.X_Byte_3);
{endregion}
			   
{region " SIGNAL AREA : NAME->X_Opp_Dist_Bat LENGTH->16 STARTBIT :32"}
_FB_UNPACK_WORD_TO_BYTE_13 (
		X_WORD_0									:= 
(*SELECT 1 : Is data valid and range is not exceed?*)	SEL((GVL.IOVD.X_Opp_Dist_Bat.v AND NOT GVL.IOVD.X_Opp_Dist_Bat.RangeExcd),
(*SELECT 2 : Is NOT AVAILABLE ?*)						SEL(GVL.IOVD.X_Opp_Dist_Bat.na,
(*SELECT 3 : Is ERROR active ?*)						SEL(GVL.IOVD.X_Opp_Dist_Bat.e,
(*DEFAULT VALUE assignment*)							0,
(*ERROR is active*)										16#FEFE),
(*NOT AVAILABLE is active*)								16#FFFF),
(*Transmission is VALID*)								UINT_TO_WORD(REAL_TO_UINT((GVL.IOVD.X_Opp_Dist_Bat.x)/0.1))),
		X_BYTE_0										=> _FB_CanTx_Message_Unpack_4CC.X_Byte_4,
		X_BYTE_1										=> _FB_CanTx_Message_Unpack_4CC.X_Byte_5);
{endregion}						 

_FB_CanTx_Message_Unpack_4CC.X_Byte_6 		:= 16#FF;
_FB_CanTx_Message_Unpack_4CC.X_Byte_7 		:= 16#FF;

_FB_CanTx_Message_Unpack_4CC (		C_Enable		:= GVL.IOVD.C_En_Sayicilar_1_0X4CC,
     								Obj_CAN			:= ADR(GVL.IC.Obj_CAN0),
     								X_MsgID			:= 16#4CC,
     								Tm_CycleTime	:= TIME#1000MS,
     								N_Msg_Dlc		:= 8,
     								S_Extended		:= 0,
     								S_Sent_Ok   	=> GVL.IOVD.S_SentOk_Sayicilar_1_0X4CC);
{endregion}
//-----------------------------------------------------------------------------------------------------------------------------
//-----------------------------------------------------------------------------------------------------------------------------
{region " MESSAGE AREA :Yardimci_Tuketici_Enerjileri- ID:4CD"}

{region " SIGNAL AREA : NAME->X_E_Aux_Cons LENGTH->32 STARTBIT :0"}
_FB_UNPACK_DWORD_TO_BYTE_16 (
		X_DWORD_0									:= 
(*SELECT 1 : Is data valid and range is not exceed?*)	SEL((GVL.IOVD.X_E_Aux_Cons.v AND NOT GVL.IOVD.X_E_Aux_Cons.RangeExcd),
(*SELECT 2 : Is NOT AVAILABLE ?*)						SEL(GVL.IOVD.X_E_Aux_Cons.na,
(*SELECT 3 : Is ERROR active ?*)						SEL(GVL.IOVD.X_E_Aux_Cons.e,
(*DEFAULT VALUE assignment*)							0,
(*ERROR is active*)										16#FEFEFEFE),
(*NOT AVAILABLE is active*)								16#FFFFFFFF),
(*Transmission is VALID*)								UDINT_TO_DWORD(REAL_TO_UDINT((GVL.IOVD.X_E_Aux_Cons.x)/0.1))),
		X_BYTE_0										=> _FB_CanTx_Message_Unpack_4CD.X_Byte_0,
		X_BYTE_1										=> _FB_CanTx_Message_Unpack_4CD.X_Byte_1,
		X_BYTE_2										=> _FB_CanTx_Message_Unpack_4CD.X_Byte_2,
		X_BYTE_3										=> _FB_CanTx_Message_Unpack_4CD.X_Byte_3);
{endregion}

{region " SIGNAL AREA : NAME->X_E_Aux_Hvac_Cons LENGTH->32 STARTBIT :32"}
_FB_UNPACK_DWORD_TO_BYTE_17 (
		X_DWORD_0									:= 
(*SELECT 1 : Is data valid and range is not exceed?*)	SEL((GVL.IOVD.X_E_Aux_Hvac_Cons.v AND NOT GVL.IOVD.X_E_Aux_Hvac_Cons.RangeExcd),
(*SELECT 2 : Is NOT AVAILABLE ?*)						SEL(GVL.IOVD.X_E_Aux_Hvac_Cons.na,
(*SELECT 3 : Is ERROR active ?*)						SEL(GVL.IOVD.X_E_Aux_Hvac_Cons.e,
(*DEFAULT VALUE assignment*)							0,
(*ERROR is active*)										16#FEFEFEFE),
(*NOT AVAILABLE is active*)								16#FFFFFFFF),
(*Transmission is VALID*)								UDINT_TO_DWORD(REAL_TO_UDINT((GVL.IOVD.X_E_Aux_Hvac_Cons.x)/0.1))),
		X_BYTE_0										=> _FB_CanTx_Message_Unpack_4CD.X_Byte_4,
		X_BYTE_1										=> _FB_CanTx_Message_Unpack_4CD.X_Byte_5,
		X_BYTE_2										=> _FB_CanTx_Message_Unpack_4CD.X_Byte_6,
		X_BYTE_3										=> _FB_CanTx_Message_Unpack_4CD.X_Byte_7);
{endregion}

_FB_CanTx_Message_Unpack_4CD (		C_Enable		:= GVL.IOVD.C_En_Yardimci_Tuketici_Enerjileri_0X4CD,
     								Obj_CAN			:= ADR(GVL.IC.Obj_CAN0),
     								X_MsgID			:= 16#4CD,
     								Tm_CycleTime	:= TIME#1000MS,
     								N_Msg_Dlc		:= 8,
     								S_Extended		:= 0,
     								S_Sent_Ok   	=> GVL.IOVD.S_SentOk_Yardimci_Tuketici_Enerjileri_0X4CD);
{endregion}
	 //-----------------------------------------------------------------------------------------------------------------------------
{region " MESSAGE AREA :Kapi_Sayicilari_1- ID:4CD"}

{region " SIGNAL AREA : NAME->N_Dr1_Cycle LENGTH->32 STARTBIT :0"}
_FB_UNPACK_DWORD_TO_BYTE_20 (
		X_DWORD_0									:= 
(*SELECT 1 : Is force active?*)							SEL((GVL.IOVD.N_Dr1_Cycle.v AND NOT GVL.IOVD.N_Dr1_Cycle.RangeExcd),
(*DEFAULT VALUE assignment*)							0,
(*FORCE is active*)										UDINT_TO_DWORD(REAL_TO_UDINT(GVL.IOVD.N_Dr1_Cycle.x))),
		X_BYTE_0										=> _FB_CanTx_Message_4CE.X_Byte_0,
		X_BYTE_1										=> _FB_CanTx_Message_4CE.X_Byte_1,
		X_BYTE_2										=> _FB_CanTx_Message_4CE.X_Byte_2,
		X_BYTE_3										=> _FB_CanTx_Message_4CE.X_Byte_3);
{endregion}
{region " SIGNAL AREA : NAME->N_Dr2_Cycle LENGTH->32 STARTBIT :32"}
_FB_UNPACK_DWORD_TO_BYTE_19 (
		X_DWORD_0									:= 
(*SELECT 1 : Is force active?*)							SEL((GVL.IOVD.N_Dr2_Cycle.v AND NOT GVL.IOVD.N_Dr2_Cycle.RangeExcd),
(*DEFAULT VALUE assignment*)							0,
(*FORCE is active*)										UDINT_TO_DWORD(REAL_TO_UDINT(GVL.IOVD.N_Dr2_Cycle.x))),
		X_BYTE_0										=> _FB_CanTx_Message_4CE.X_Byte_4,
		X_BYTE_1										=> _FB_CanTx_Message_4CE.X_Byte_5,
		X_BYTE_2										=> _FB_CanTx_Message_4CE.X_Byte_6,
		X_BYTE_3										=> _FB_CanTx_Message_4CE.X_Byte_7);
{endregion}

_FB_CanTx_Message_4CE (		C_Enable		:= GVL.IOVD.C_En_Kapi_Sayicilari_1_0X4CE,
     						Obj_CAN			:= ADR(GVL.IC.Obj_CAN0),
     						X_MsgID			:= 16#4CE,
     						Tm_CycleTime	:= TIME#1000MS,
     						N_Msg_Dlc		:= 8,
     						S_Extended		:= 0,
     						S_Sent_Ok   	=> GVL.IOVD.S_SentOk_Kapi_Sayicilari_1_0X4CE);
{endregion}
//-----------------------------------------------------------------------------------------------------------------------------
//-----------------------------------------------------------------------------------------------------------------------------
{region " MESSAGE AREA :Kapi_Sayicilari_2- ID:4CF"}

{region " SIGNAL AREA : NAME->N_Dr3_Cycle LENGTH->32 STARTBIT :0"}
_FB_UNPACK_DWORD_TO_BYTE_22 (
		X_DWORD_0									:= 
(*SELECT 1 : Is force active?*)							SEL((GVL.IOVD.N_Dr3_Cycle.v AND NOT GVL.IOVD.N_Dr3_Cycle.RangeExcd),
(*DEFAULT VALUE assignment*)							0,
(*FORCE is active*)										UDINT_TO_DWORD(REAL_TO_UDINT(GVL.IOVD.N_Dr3_Cycle.x))),
		X_BYTE_0										=> _FB_CanTx_Message_4CF.X_Byte_0,
		X_BYTE_1										=> _FB_CanTx_Message_4CF.X_Byte_1,
		X_BYTE_2										=> _FB_CanTx_Message_4CF.X_Byte_2,
		X_BYTE_3										=> _FB_CanTx_Message_4CF.X_Byte_3);
{endregion}
{region " SIGNAL AREA : NAME->N_Dr4_Cycle LENGTH->32 STARTBIT :32"}
_FB_UNPACK_DWORD_TO_BYTE_21 (
		X_DWORD_0									:= 
(*SELECT 1 : Is force active?*)							SEL((GVL.IOVD.N_Dr4_Cycle.v AND NOT GVL.IOVD.N_Dr4_Cycle.RangeExcd),
(*DEFAULT VALUE assignment*)							0,
(*FORCE is active*)										UDINT_TO_DWORD(REAL_TO_UDINT(GVL.IOVD.N_Dr4_Cycle.x))),
		X_BYTE_0										=> _FB_CanTx_Message_4CF.X_Byte_4,
		X_BYTE_1										=> _FB_CanTx_Message_4CF.X_Byte_5,
		X_BYTE_2										=> _FB_CanTx_Message_4CF.X_Byte_6,
		X_BYTE_3										=> _FB_CanTx_Message_4CF.X_Byte_7);
{endregion}

_FB_CanTx_Message_4CF (		C_Enable		:= GVL.IOVD.C_En_Kapi_Sayicilari_2_0X4CF,
     						Obj_CAN			:= ADR(GVL.IC.Obj_CAN0),
     						X_MsgID			:= 16#4CF,
     						Tm_CycleTime	:= TIME#1000MS,
     						N_Msg_Dlc		:= 8,
     						S_Extended		:= 0,
     						S_Sent_Ok   	=> GVL.IOVD.S_SentOk_Kapi_Sayicilari_2_0X4CF);
{endregion}
//-----------------------------------------------------------------------------------------------------------------------------
//-----------------------------------------------------------------------------------------------------------------------------
{region " MESSAGE AREA :Sarj_Enerjisi- ID:4D0"}

{region " SIGNAL AREA : NAME->X_E_Chrg_Onbrd LENGTH->32 STARTBIT :0"}
_FB_UNPACK_DWORD_TO_BYTE_24 (
		X_DWORD_0									:= 
(*SELECT 1 : Is force active?*)							SEL((GVL.IOVD.X_E_Chrg_Onbrd.v AND NOT GVL.IOVD.X_E_Chrg_Onbrd.RangeExcd),
(*DEFAULT VALUE assignment*)							0,
(*FORCE is active*)										UDINT_TO_DWORD(REAL_TO_UDINT((GVL.IOVD.X_E_Chrg_Onbrd.x)/0.1))),
		X_BYTE_0										=> _FB_CanTx_Message_4D0.X_Byte_0,
		X_BYTE_1										=> _FB_CanTx_Message_4D0.X_Byte_1,
		X_BYTE_2										=> _FB_CanTx_Message_4D0.X_Byte_2,
		X_BYTE_3										=> _FB_CanTx_Message_4D0.X_Byte_3);
{endregion}
{region " SIGNAL AREA : NAME->X_E_Chrg_Pan LENGTH->32 STARTBIT :32"}
_FB_UNPACK_DWORD_TO_BYTE_23 (
		X_DWORD_0									:= 
(*SELECT 1 : Is force active?*)							SEL((GVL.IOVD.X_E_Chrg_Pan.v AND NOT GVL.IOVD.X_E_Chrg_Pan.RangeExcd),
(*DEFAULT VALUE assignment*)							0,
(*FORCE is active*)										UDINT_TO_DWORD(REAL_TO_UDINT((GVL.IOVD.X_E_Chrg_Pan.x)/0.1))),
		X_BYTE_0										=> _FB_CanTx_Message_4D0.X_Byte_4,
		X_BYTE_1										=> _FB_CanTx_Message_4D0.X_Byte_5,
		X_BYTE_2										=> _FB_CanTx_Message_4D0.X_Byte_6,
		X_BYTE_3										=> _FB_CanTx_Message_4D0.X_Byte_7);
{endregion}

_FB_CanTx_Message_4D0 (		C_Enable		:= GVL.IOVD.C_En_Sarj_Enerjisi_0X4D0,
     						Obj_CAN			:= ADR(GVL.IC.Obj_CAN0),
     						X_MsgID			:= 16#4D0,
     						Tm_CycleTime	:= TIME#1000MS,
     						N_Msg_Dlc		:= 8,
     						S_Extended		:= 0,
     						S_Sent_Ok  		=> GVL.IOVD.S_SentOk_Sarj_Enerjisi_0X4D0);
{endregion}
//-----------------------------------------------------------------------------------------------------------------------------
//-----------------------------------------------------------------------------------------------------------------------------
//-----------------------------------------------------------------------------------------------------------------------------
{region " MESSAGE AREA :Arac_Bilgi_1- ID:4E0"}

{region " SIGNAL AREA : NAME->X_Vh_No LENGTH->16 STARTBIT :0"}
_FB_UNPACK_WORD_TO_BYTE_11 (
		X_WORD_0									:= 
(*SELECT 1 : Is data valid and range is not exceed?*)	SEL((GVL.IOVD.X_Vh_No.v AND NOT GVL.IOVD.X_Vh_No.RangeExcd),
(*SELECT 2 : Is NOT AVAILABLE ?*)						SEL(GVL.IOVD.X_Vh_No.na,
(*SELECT 3 : Is ERROR active ?*)						SEL(GVL.IOVD.X_Vh_No.e,
(*DEFAULT VALUE assignment*)							0,
(*ERROR is active*)										16#FEFE),
(*NOT AVAILABLE is active*)								16#FFFF),
(*Transmission is VALID*)								UINT_TO_WORD(REAL_TO_UINT((GVL.IOVD.X_Vh_No.x)))),
		X_BYTE_0										=> _FB_CanTx_Message_4E0.X_Byte_0,
		X_BYTE_1										=> _FB_CanTx_Message_4E0.X_Byte_1);

{endregion}

{region " SIGNAL AREA : NAME->X_Sw_Ver_Mjr_ECU LENGTH->8 STARTBIT :16"}
_FB_CanTx_Message_4E0.X_Byte_2						:=
(*SELECT 1 : Is data valid and range is not exceed?*)	SEL((GVL.IOVD.X_Sw_Ver_Mjr_ECU.v AND NOT GVL.IOVD.X_Sw_Ver_Mjr_ECU.RangeExcd),
(*SELECT 2 : Is NOT AVAILABLE ?*)						SEL(GVL.IOVD.X_Sw_Ver_Mjr_ECU.na,
(*SELECT 3 : Is ERROR active ?*)						SEL(GVL.IOVD.X_Sw_Ver_Mjr_ECU.e,
(*DEFAULT VALUE assignment*)							0,
(*ERROR is active*)										16#FE),
(*NOT AVAILABLE is active*)								16#FF),
(*Transmission is VALID*)								USINT_TO_BYTE(REAL_TO_USINT((GVL.IOVD.X_Sw_Ver_Mjr_ECU.x))));
{endregion}

{region " SIGNAL AREA : NAME->X_Sw_Ver_Mnr_ECU LENGTH->8 STARTBIT :24"}
_FB_CanTx_Message_4E0.X_Byte_3						:=
(*SELECT 1 : Is data valid and range is not exceed?*)	SEL((GVL.IOVD.X_Sw_Ver_Mnr_ECU.v AND NOT GVL.IOVD.X_Sw_Ver_Mnr_ECU.RangeExcd),
(*SELECT 2 : Is NOT AVAILABLE ?*)						SEL(GVL.IOVD.X_Sw_Ver_Mnr_ECU.na,
(*SELECT 3 : Is ERROR active ?*)						SEL(GVL.IOVD.X_Sw_Ver_Mnr_ECU.e,
(*DEFAULT VALUE assignment*)							0,
(*ERROR is active*)										16#FE),
(*NOT AVAILABLE is active*)								16#FF),
(*Transmission is VALID*)								USINT_TO_BYTE(REAL_TO_USINT((GVL.IOVD.X_Sw_Ver_Mnr_ECU.x))));
{endregion}

{region " SIGNAL AREA : NAME->X_Sw_Ver_Tst_ECU LENGTH->8 STARTBIT :32"}
_FB_CanTx_Message_4E0.X_Byte_4						:=
(*SELECT 1 : Is data valid and range is not exceed?*)	SEL((GVL.IOVD.X_Sw_Ver_Tst_ECU.v AND NOT GVL.IOVD.X_Sw_Ver_Tst_ECU.RangeExcd),
(*SELECT 2 : Is NOT AVAILABLE ?*)						SEL(GVL.IOVD.X_Sw_Ver_Tst_ECU.na,
(*SELECT 3 : Is ERROR active ?*)						SEL(GVL.IOVD.X_Sw_Ver_Tst_ECU.e,
(*DEFAULT VALUE assignment*)							0,
(*ERROR is active*)										16#FE),
(*NOT AVAILABLE is active*)								16#FF),
(*Transmission is VALID*)								USINT_TO_BYTE(REAL_TO_USINT((GVL.IOVD.X_Sw_Ver_Tst_ECU.x))));
{endregion}

{region " SIGNAL AREA : NAME->X_Sw_Ver_Mjr_TCU LENGTH->8 STARTBIT :24"}
_FB_CanTx_Message_4E0.X_Byte_5						:=
(*SELECT 1 : Is data valid and range is not exceed?*)	SEL((GVL.IOVD.X_Sw_Ver_Mjr_TCU.v AND NOT GVL.IOVD.X_Sw_Ver_Mjr_TCU.RangeExcd),
(*SELECT 2 : Is NOT AVAILABLE ?*)						SEL(GVL.IOVD.X_Sw_Ver_Mjr_TCU.na,
(*SELECT 3 : Is ERROR active ?*)						SEL(GVL.IOVD.X_Sw_Ver_Mjr_TCU.e,
(*DEFAULT VALUE assignment*)							0,
(*ERROR is active*)										16#FE),
(*NOT AVAILABLE is active*)								16#FF),
(*Transmission is VALID*)								USINT_TO_BYTE(REAL_TO_USINT((GVL.IOVD.X_Sw_Ver_Mjr_TCU.x))));
{endregion}
		  
{region " SIGNAL AREA : NAME->X_Sw_Ver_Mnr_TCU LENGTH->8 STARTBIT :32"}
_FB_CanTx_Message_4E0.X_Byte_6						:=
(*SELECT 1 : Is data valid and range is not exceed?*)	SEL((GVL.IOVD.X_Sw_Ver_Mnr_TCU.v AND NOT GVL.IOVD.X_Sw_Ver_Mnr_TCU.RangeExcd),
(*SELECT 2 : Is NOT AVAILABLE ?*)						SEL(GVL.IOVD.X_Sw_Ver_Mnr_TCU.na,
(*SELECT 3 : Is ERROR active ?*)						SEL(GVL.IOVD.X_Sw_Ver_Mnr_TCU.e,
(*DEFAULT VALUE assignment*)							0,
(*ERROR is active*)										16#FE),
(*NOT AVAILABLE is active*)								16#FF),
(*Transmission is VALID*)								USINT_TO_BYTE(REAL_TO_USINT((GVL.IOVD.X_Sw_Ver_Mnr_TCU.x))));
{endregion}
		
{region " SIGNAL AREA : NAME->X_Sw_Ver_Tst_TCU LENGTH->8 STARTBIT :40"}
_FB_CanTx_Message_4E0.X_Byte_7						:=
(*SELECT 1 : Is data valid and range is not exceed?*)	SEL((GVL.IOVD.X_Sw_Ver_Tst_TCU.v AND NOT GVL.IOVD.X_Sw_Ver_Tst_TCU.RangeExcd),
(*SELECT 2 : Is NOT AVAILABLE ?*)						SEL(GVL.IOVD.X_Sw_Ver_Tst_TCU.na,
(*SELECT 3 : Is ERROR active ?*)						SEL(GVL.IOVD.X_Sw_Ver_Tst_TCU.e,
(*DEFAULT VALUE assignment*)							0,
(*ERROR is active*)										16#FE),
(*NOT AVAILABLE is active*)								16#FF),
(*Transmission is VALID*)								USINT_TO_BYTE(REAL_TO_USINT((GVL.IOVD.X_Sw_Ver_Tst_TCU.x))));
{endregion}
					
_FB_CanTx_Message_4E0 (		C_Enable		:= GVL.IOVD.C_En_Arac_Bilgi_1_0X4E0,
     						Obj_CAN			:= ADR(GVL.IC.Obj_CAN0),
     						X_MsgID			:= 16#4E0,
     						Tm_CycleTime	:= TIME#5000MS,
     						N_Msg_Dlc		:= 8,
     						S_Extended		:= 0,
     						S_Sent_Ok   	=> GVL.IOVD.S_SentOk_Arac_Bilgi_1_0X4E0);
{endregion}
//-----------------------------------------------------------------------------------------------------------------------------
//-----------------------------------------------------------------------------------------------------------------------------
//-----------------------------------------------------------------------------------------------------------------------------


                  
END_PROGRAM

FUNCTION_BLOCK _FB_Time_Get
  VAR_INPUT
    C_Set_Time : BOOL;  (* Command to set new time *)
    Obj_Time : XTime_T;  (* Assign that the time comes from diagnose *)
    Adr_Obj_Time : POINTER TO XTime_T;  (* System time variables *)
  END_VAR
  VAR_OUTPUT
    Tm_SystemRuntime : TIME;  (* System runtime 24h cycle *)
    ER_RTC_MssRead : BOOL;  (* Runtime calculation is failed because of RTC register is not increasing the time *)
  END_VAR
  VAR
    S_Init : BOOL := TRUE;
    S_Sys_Time_Read_En : lib500_types.IO_ERRORTYPE := lib500_types.IO_ERRORTYPE.IO_E_OK;
    S_Set_Time_Old : BOOL;
    S_Set_Time_Act : BOOL;
    S_Set_New_Det : BOOL;
    X_Cont_TmStartup_Ms : DWORD;
    X_Cont_TmActual_Ms : DWORD;
    X_Cont_SystemRuntime : DWORD;
  END_VAR

                    
IF(S_Sys_Time_Read_En <> lib500_types.IO_ERRORTYPE.IO_E_BUSY) THEN
	S_Sys_Time_Read_En := lib500.IO_RTC_GetDateAndTime(ADR(Adr_Obj_Time^.X_Seconds),(Adr_Obj_Time^.X_Minutes),(Adr_Obj_Time^.X_Hours),(Adr_Obj_Time^.X_Days),(Adr_Obj_Time^.X_Months),(Adr_Obj_Time^.X_Years));
END_IF

X_Cont_TmActual_Ms := BYTE_TO_DWORD(Adr_Obj_Time^.X_Seconds * 100) + BYTE_TO_DWORD(Adr_Obj_Time^.X_Minutes*60*100) + BYTE_TO_DWORD(Adr_Obj_Time^.X_Hours * 60 * 60 * 100);
S_Set_Time_Act := C_Set_Time;

IF(S_Set_Time_Act <> S_Set_Time_Old) THEN
	IF S_Set_Time_Act THEN
		S_Set_New_Det := TRUE;
	END_IF
   	S_Set_Time_Old := S_Set_Time_Act;
END_IF

IF(S_Init OR S_Set_New_Det) THEN
	S_Sys_Time_Read_En := lib500.IO_RTC_InitDateAndTime();
	S_Sys_Time_Read_En := lib500.IO_RTC_GetDateAndTime(Obj_Time.X_Seconds,Obj_Time.X_Minutes,Obj_Time.X_Hours,Obj_Time.X_Days,Obj_Time.X_Months,Obj_Time.X_Years);
	X_Cont_TmStartup_Ms := X_Cont_TmActual_Ms ;
	IF S_Init THEN
		S_Init := FALSE;
	END_IF
	S_Set_New_Det := FALSE;
END_IF

S_Sys_Time_Read_En:=lib500.IO_RTC_GetDateAndTimeStatus();

IF(X_Cont_TmActual_Ms > X_Cont_TmStartup_Ms) THEN
	Tm_SystemRuntime := DWORD_TO_TIME(X_Cont_TmActual_Ms - X_Cont_TmStartup_Ms);
	ER_RTC_MssRead := FALSE;
ELSE	
	IF NOT ER_RTC_MssRead THEN
	X_Cont_TmStartup_Ms := X_Cont_TmActual_Ms;
	END_IF
	ER_RTC_MssRead := TRUE;
END_IF

                  
END_FUNCTION_BLOCK

FUNCTION_BLOCK _FB_Tools_Dir_Prop
  VAR_INPUT
    X_Act_Val : REAL;
    X_Min_Lim : REAL;
    X_Max_Lim : REAL;
  END_VAR
  VAR_OUTPUT
    X_Der_Pct : REAL;
  END_VAR

                    IF X_Min_Lim >= X_Max_Lim THEN
	X_Der_Pct := 0;
ELSE
	IF X_Act_Val <= X_Min_Lim THEN
		X_Der_Pct := 0;
	ELSIF X_Act_Val >= X_Max_Lim THEN
		X_Der_Pct := 100;
	ELSE
		X_Der_Pct := ((X_Act_Val - X_Min_Lim) * 100) / (X_Max_Lim - X_Min_Lim);
	END_IF
END_IF

IF X_Der_Pct > 100 THEN
	X_Der_Pct := 100;
END_IF
                  
END_FUNCTION_BLOCK

FUNCTION_BLOCK _FB_Tools_Inv_Prop
  VAR_INPUT
    X_Act_Val : REAL;
    X_Min_Lim : REAL;
    X_Max_Lim : REAL;
  END_VAR
  VAR_OUTPUT
    X_Der_Pct : REAL;
  END_VAR

                    IF X_Min_Lim >= X_Max_Lim THEN
	
	X_Der_Pct := 0;
	
ELSE
	
	IF X_Act_Val <= X_Min_Lim THEN
		X_Der_Pct := 100;
	ELSIF X_Act_Val >= X_Max_Lim THEN
		X_Der_Pct := 0;
	ELSE
		X_Der_Pct := ((X_Max_Lim - X_Act_Val) * 100) / (X_Max_Lim - X_Min_Lim);
	END_IF

END_IF

IF X_Der_Pct > 100 THEN
	
	X_Der_Pct := 100;
	
END_IF
                  
END_FUNCTION_BLOCK

FUNCTION_BLOCK UdpSocket
  VAR
    hSocket : RTS_IEC_HANDLE := RTS_INVALID_HANDLE;  (* Handle to the socket *)
  END_VAR

                    
                  

METHOD SendTo : __XINT
  VAR_INPUT
    pbyBuffer : POINTER TO BYTE;  (* Buffer with send data *)
    diBufferSize : __XINT;  (* Length OF data TO send *)
    diFlags : DINT;  (* Flags parameter *)
    pSockAddr : POINTER TO SOCKADDRESS;  (* Socket address AND port TO sent data TO *)
    diSockAddrSize : DINT;  (* Size OF socket address structure *)
    pResult : POINTER TO RTS_IEC_RESULT;  (* POINTER TO runtime system error code (see CmpErrors.library) *)
  END_VAR
                          // check, if this instance has been initialized
IF (THIS^.hSocket <> RTS_INVALID_HANDLE) THEN
	SendTo := SysSocket.SysSockSendTo(THIS^.hSocket, pbyBuffer, diBufferSize, diFlags, pSockAddr, diSockAddrSize, pResult);
END_IF
                        
END_METHOD

METHOD RecvFrom : __XINT
  VAR_INPUT
    pbyBuffer : POINTER TO BYTE;  (* Buffer; TO read data FROM the socket *)
    diBufferSize : __XINT;  (* Maximum length OF the buffer *)
    diFlags : DINT;  (* Flags parameter *)
    pSockAddr : POINTER TO SOCKADDRESS;  (* Socket address AND port TO receive data FROM *)
    diSockAddrSize : DINT;  (* Size OF socket address structure *)
    pResult : POINTER TO RTS_IEC_RESULT;  (* POINTER TO runtime system error code (see CmpErrors.library) *)
  END_VAR
                          // check, if this instance has been initialized
IF (THIS^.hSocket <> RTS_INVALID_HANDLE) THEN
	RecvFrom := SysSocket.SysSockRecvFrom(THIS^.hSocket, pbyBuffer, diBufferSize, diFlags, pSockAddr, diSockAddrSize, pResult);
END_IF
                        
END_METHOD

METHOD Bind : RTS_IEC_HANDLE
  VAR_INPUT
    pSockAddr : POINTER TO SOCKADDRESS;  (* Socket address *)
    diSockAddrSize : DINT;  (* Size of the socket address structure *)
  END_VAR
                          // check, if this instance has been initialized
IF (THIS^.hSocket <> RTS_INVALID_HANDLE) THEN
	Bind := SysSockBind(THIS^.hSocket, pSockAddr, diSockAddrSize);
END_IF
                        
END_METHOD

METHOD FB_exit : BOOL
  VAR_INPUT
    bInCopyCode : BOOL;
  END_VAR
                          // check, for a previous initialization of this instance
IF (THIS^.hSocket <> RTS_INVALID_HANDLE) THEN
	// perform automatic closing
	SysSocket.SysSockClose(THIS^.hSocket);
END_IF
                        
END_METHOD

